	(*-------------- Services Stand EtherCAT Slave Faults----------------------------*)
	(*Fault584 - EtherCAT Slave Fault on Services Stand 01*)
		Fault_Tmrs[584].PT:= No_Timer;
		Fault_Tmrs[584]();
		Fault_Tmrs[584].IN:= GTAC_CONFIG.Option_Air1 AND NOT MAIN.SS01.DiscreteNode_OK;
		Out_To_ICxx.System_Faults[584]:=Fault_Tmrs[584].Q;
	(*Fault585 - EtherCAT Slave Fault on Services Stand 02*)
		Fault_Tmrs[585].PT:= No_Timer;
		Fault_Tmrs[585]();
		Fault_Tmrs[585].IN:= GTAC_CONFIG.Option_Air2 AND NOT MAIN.SS02.DiscreteNode_OK;
		Out_To_ICxx.System_Faults[585]:=Fault_Tmrs[585].Q;
	(*Fault586 - EtherCAT Slave Fault on Services Stand 03*)
		Fault_Tmrs[586].PT:= No_Timer;
		Fault_Tmrs[586]();
		Fault_Tmrs[586].IN:= FALSE AND NOT MAIN.SS03.DiscreteNode_OK;
		Out_To_ICxx.System_Faults[586]:=Fault_Tmrs[586].Q;

	(*-------------- Enable Switch Plate EtherCAT Slave Faults----------------------------*)
	(*Fault587 - EtherCAT Slave Fault on Enable Switch Plate 01*)
		Fault_Tmrs[587].PT:= No_Timer;
		Fault_Tmrs[587]();
		Fault_Tmrs[587].IN:= (GTAC_CONFIG.Option_ESW_Count>=1)
							AND NOT MAIN.ESW01.DiscreteNode_OK;
		Out_To_ICxx.System_Faults[587]:=Fault_Tmrs[587].Q;

	(*Fault588 - EtherCAT Slave Fault on Enable Switch Plate 02*)
		Fault_Tmrs[588].PT:= No_Timer;
		Fault_Tmrs[588]();
		Fault_Tmrs[588].IN:=  (GTAC_CONFIG.Option_ESW_Count>=2)
							 AND NOT MAIN.ESW02.DiscreteNode_OK;
		Out_To_ICxx.System_Faults[588]:=Fault_Tmrs[588].Q;

	(*Fault589 - EtherCAT Slave Fault on Enable Switch Plate 03*)
		Fault_Tmrs[589].PT:= No_Timer;
		Fault_Tmrs[589]();
		Fault_Tmrs[589].IN:=  (GTAC_CONFIG.Option_ESW_Count>=3)
							 AND NOT MAIN.ESW03.DiscreteNode_OK;
		Out_To_ICxx.System_Faults[589]:=Fault_Tmrs[589].Q;

	(*Fault590 - EtherCAT Slave Fault on Enable Switch Plate 04*)
		Fault_Tmrs[590].PT:= No_Timer;
		Fault_Tmrs[590]();
		Fault_Tmrs[590].IN:=  (GTAC_CONFIG.Option_ESW_Count>=4)
							 AND NOT MAIN.ESW04.DiscreteNode_OK;
		Out_To_ICxx.System_Faults[590]:=Fault_Tmrs[590].Q;

	(*-----------------ICxx EtherCAT Slave Faulted--------------*)

	(*Fault591 - EtherCAT Slave Fault In IC01 Cabinet*)
		Fault_Tmrs[591].PT:= No_Timer;
		Fault_Tmrs[591]();
		Fault_Tmrs[591].IN:= (GTAC_CONFIG.Option_IC_Count>=1) AND
							NOT MAIN.IC01.DiscreteNode_OK;
		Out_To_ICxx.System_Faults[591]:=Fault_Tmrs[591].Q;
	(*Fault592 - EtherCAT Slave Fault In IC02 Cabinet*)
		Fault_Tmrs[592].PT:= No_Timer;
		Fault_Tmrs[592]();
		Fault_Tmrs[592].IN:= (GTAC_CONFIG.Option_IC_Count>=2) AND
							NOT MAIN.IC02.DiscreteNode_OK;
		Out_To_ICxx.System_Faults[592]:=Fault_Tmrs[592].Q;
	(*Fault593 - EtherCAT Slave Fault In IC03 Cabinet*)
		Fault_Tmrs[593].PT:= No_Timer;
		Fault_Tmrs[593]();
		Fault_Tmrs[593].IN:= (GTAC_CONFIG.Option_IC_Count>=3) AND
							NOT MAIN.IC03.DiscreteNode_OK;
		Out_To_ICxx.System_Faults[593]:=Fault_Tmrs[593].Q;
	(*Fault594 - EtherCAT Slave Fault In IC04 Cabinet*)
		Fault_Tmrs[594].PT:= No_Timer;
		Fault_Tmrs[594]();
		Fault_Tmrs[594].IN:= (GTAC_CONFIG.Option_IC_Count>=4) AND
							NOT MAIN.IC04.DiscreteNode_OK;
		Out_To_ICxx.System_Faults[594]:=Fault_Tmrs[594].Q;
	(*Fault595 - EtherCAT Slave Fault In IC05 Cabinet*)
		Fault_Tmrs[595].PT:= No_Timer;
		Fault_Tmrs[595]();
		Fault_Tmrs[595].IN:= (GTAC_CONFIG.Option_IC_Count>=5) AND
							NOT MAIN.IC05.DiscreteNode_OK;
		Out_To_ICxx.System_Faults[595]:=Fault_Tmrs[595].Q;
	(*Fault596 - EtherCAT Slave Fault In IC06 Cabinet*)
		Fault_Tmrs[596].PT:= No_Timer;
		Fault_Tmrs[596]();
		Fault_Tmrs[596].IN:= (GTAC_CONFIG.Option_IC_Count>=6) AND
							NOT MAIN.IC06.DiscreteNode_OK;
		Out_To_ICxx.System_Faults[596]:=Fault_Tmrs[596].Q;
	(*Fault597 - EtherCAT Slave Fault In IC07 Cabinet*)
		Fault_Tmrs[597].PT:= No_Timer;
		Fault_Tmrs[597]();
		Fault_Tmrs[597].IN:= (GTAC_CONFIG.Option_IC_Count>=7) AND
							NOT MAIN.IC07.DiscreteNode_OK;
		Out_To_ICxx.System_Faults[597]:=Fault_Tmrs[597].Q;
	(*Fault598 - EtherCAT Slave Fault In IC08 Cabinet*)
		Fault_Tmrs[598].PT:= No_Timer;
		Fault_Tmrs[598]();
		Fault_Tmrs[598].IN:= (GTAC_CONFIG.Option_IC_Count>=8) AND
							NOT MAIN.IC08.DiscreteNode_OK;
		Out_To_ICxx.System_Faults[598]:=Fault_Tmrs[598].Q;

	(*------------------------------------------------- Fix_XX EtherCAT Slave Faults --------------------------------------------------*)

	(*IC related Fixtures (Human)*)
	(*Fault601 - EtherCAT Slave Fault On Fix at IC01.OP1*)
		Fault_Tmrs[601].PT:= No_Timer;
		Fault_Tmrs[601]();
		Fault_Tmrs[601].IN:= GTAC_CONFIG.Option_HumanFix_Enables.1 AND
							NOT Fix01.DiscreteNode_OK;
		Out_To_ICxx.System_Faults[601]:=Fault_Tmrs[601].Q;
	(*Fault602 - EtherCAT Slave Fault On Fix at IC01.OP2*)
		Fault_Tmrs[602].PT:= No_Timer;
		Fault_Tmrs[602]();
		Fault_Tmrs[602].IN:= GTAC_CONFIG.Option_HumanFix_Enables.2 AND
							NOT Fix02.DiscreteNode_OK;
		Out_To_ICxx.System_Faults[602]:=Fault_Tmrs[602].Q;

	(*Fault603 - EtherCAT Slave Fault On Fix at IC02.OP1*)
		Fault_Tmrs[603].PT:= No_Timer;
		Fault_Tmrs[603]();
		Fault_Tmrs[603].IN:= GTAC_CONFIG.Option_HumanFix_Enables.3 AND
							NOT Fix03.DiscreteNode_OK;
		Out_To_ICxx.System_Faults[603]:=Fault_Tmrs[603].Q;
	(*Fault604 - EtherCAT Slave Fault On Fix at IC02.OP2*)
		Fault_Tmrs[604].PT:= No_Timer;
		Fault_Tmrs[604]();
		Fault_Tmrs[604].IN:= GTAC_CONFIG.Option_HumanFix_Enables.4 AND
							NOT Fix04.DiscreteNode_OK;
		Out_To_ICxx.System_Faults[604]:=Fault_Tmrs[604].Q;

	(*Fault605 - EtherCAT Slave Fault On Fix at IC03.OP1*)
		Fault_Tmrs[605].PT:= No_Timer;
		Fault_Tmrs[605]();
		Fault_Tmrs[605].IN:= GTAC_CONFIG.Option_HumanFix_Enables.5 AND
							NOT Fix05.DiscreteNode_OK;
		Out_To_ICxx.System_Faults[605]:=Fault_Tmrs[605].Q;
	(*Fault606 - EtherCAT Slave Fault On Fix at IC03.OP2*)
		Fault_Tmrs[606].PT:= No_Timer;
		Fault_Tmrs[606]();
		Fault_Tmrs[606].IN:= GTAC_CONFIG.Option_HumanFix_Enables.6 AND
							NOT Fix06.DiscreteNode_OK;
		Out_To_ICxx.System_Faults[606]:=Fault_Tmrs[606].Q;

	(*Fault607 - EtherCAT Slave Fault On Fix at IC04.OP1*)
		Fault_Tmrs[607].PT:= No_Timer;
		Fault_Tmrs[607]();
		Fault_Tmrs[607].IN:= GTAC_CONFIG.Option_HumanFix_Enables.7 AND
							NOT Fix07.DiscreteNode_OK;
		Out_To_ICxx.System_Faults[607]:=Fault_Tmrs[607].Q;
	(*Fault608 - EtherCAT Slave Fault On Fix at IC04.OP2*)
		Fault_Tmrs[608].PT:= No_Timer;
		Fault_Tmrs[608]();
		Fault_Tmrs[608].IN:= GTAC_CONFIG.Option_HumanFix_Enables.8 AND
							NOT Fix08.DiscreteNode_OK;
		Out_To_ICxx.System_Faults[608]:=Fault_Tmrs[608].Q;

	(*Fault609 - EtherCAT Slave Fault On Fix at IC05.OP1*)
		Fault_Tmrs[609].PT:= No_Timer;
		Fault_Tmrs[609]();
		Fault_Tmrs[609].IN:= GTAC_CONFIG.Option_HumanFix_Enables.9 AND
							NOT Fix09.DiscreteNode_OK;
		Out_To_ICxx.System_Faults[609]:=Fault_Tmrs[609].Q;
	(*Fault610 - EtherCAT Slave Fault On Fix at IC05.OP2*)
		Fault_Tmrs[610].PT:= No_Timer;
		Fault_Tmrs[610]();
		Fault_Tmrs[610].IN:= GTAC_CONFIG.Option_HumanFix_Enables.10 AND
							NOT Fix10.DiscreteNode_OK;
		Out_To_ICxx.System_Faults[610]:=Fault_Tmrs[610].Q;

	(*Fault611 - EtherCAT Slave Fault On Fix at IC06.OP1*)
		Fault_Tmrs[611].PT:= No_Timer;
		Fault_Tmrs[611]();
		Fault_Tmrs[611].IN:= GTAC_CONFIG.Option_HumanFix_Enables.11 AND
							 NOT Fix11.DiscreteNode_OK;
		Out_To_ICxx.System_Faults[611]:=Fault_Tmrs[611].Q;
	(*Fault612 - EtherCAT Slave Fault On Fix at IC06.OP2*)
		Fault_Tmrs[612].PT:= No_Timer;
		Fault_Tmrs[612]();
		Fault_Tmrs[612].IN:= GTAC_CONFIG.Option_HumanFix_Enables.12 AND
							NOT Fix12.DiscreteNode_OK;
		Out_To_ICxx.System_Faults[612]:=Fault_Tmrs[612].Q;

	(*Fault613 - EtherCAT Slave Fault On Fix at IC07.OP1*)
		Fault_Tmrs[613].PT:= No_Timer;
		Fault_Tmrs[613]();
		Fault_Tmrs[613].IN:= GTAC_CONFIG.Option_HumanFix_Enables.13 AND
							NOT Fix13.DiscreteNode_OK;
		Out_To_ICxx.System_Faults[613]:=Fault_Tmrs[613].Q;
	(*Fault614 - EtherCAT Slave Fault On Fix at IC07.OP2*)
		Fault_Tmrs[614].PT:= No_Timer;
		Fault_Tmrs[614]();
		Fault_Tmrs[614].IN:= GTAC_CONFIG.Option_HumanFix_Enables.14 AND
							NOT Fix14.DiscreteNode_OK;
		Out_To_ICxx.System_Faults[614]:=Fault_Tmrs[614].Q;

	(*Fault615 - EtherCAT Slave Fault On Fix at IC08.OP1*)
		Fault_Tmrs[615].PT:= No_Timer;
		Fault_Tmrs[615]();
		Fault_Tmrs[615].IN:= GTAC_CONFIG.Option_HumanFix_Enables.15 AND
							NOT Fix15.DiscreteNode_OK;
		Out_To_ICxx.System_Faults[615]:=Fault_Tmrs[615].Q;
	(*Fault616 - EtherCAT Slave Fault On Fix at IC08.OP2*)
		Fault_Tmrs[616].PT:= No_Timer;
		Fault_Tmrs[616]();
		Fault_Tmrs[616].IN:= GTAC_CONFIG.Option_HumanFix_Enables.16 AND
							NOT Fix16.DiscreteNode_OK;
		Out_To_ICxx.System_Faults[616]:=Fault_Tmrs[616].Q;

	(*Internal Fixtures*)
	(*Fault617 - EtherCAT Slave Fault On Internal Fix 101*)
		Fault_Tmrs[617].PT:= No_Timer;
		Fault_Tmrs[617]();
		Fault_Tmrs[617].IN:= (GTAC_CONFIG.Option_InternalFix_Count>=1) AND
							NOT Fix101.DiscreteNode_OK;
		Out_To_ICxx.System_Faults[617]:=Fault_Tmrs[617].Q;

	(*Fault618 - EtherCAT Slave Fault On Internal Fix 102*)
		Fault_Tmrs[618].PT:= No_Timer;
		Fault_Tmrs[618]();
		Fault_Tmrs[618].IN:= (GTAC_CONFIG.Option_InternalFix_Count>=2) AND
							NOT Fix102.DiscreteNode_OK;
		Out_To_ICxx.System_Faults[618]:=Fault_Tmrs[618].Q;

	(*Fault619 - EtherCAT Slave Fault On Internal Fix 103*)
		Fault_Tmrs[619].PT:= No_Timer;
		Fault_Tmrs[619]();
		Fault_Tmrs[619].IN:= (GTAC_CONFIG.Option_InternalFix_Count>=3) AND
							NOT Fix103.DiscreteNode_OK;
		Out_To_ICxx.System_Faults[619]:=Fault_Tmrs[619].Q;

	(*Fault620 - EtherCAT Slave Fault On Internal Fix 104*)
		Fault_Tmrs[620].PT:= No_Timer;
		Fault_Tmrs[620]();
		Fault_Tmrs[620].IN:= (GTAC_CONFIG.Option_InternalFix_Count>=4) AND
							NOT Fix104.DiscreteNode_OK;
		Out_To_ICxx.System_Faults[620]:=Fault_Tmrs[620].Q;

	(*Fault621 - EtherCAT Slave Fault On Internal Fix 105*)
		Fault_Tmrs[621].PT:= No_Timer;
		Fault_Tmrs[621]();
		Fault_Tmrs[621].IN:= (GTAC_CONFIG.Option_InternalFix_Count>=5) AND
							NOT Fix105.DiscreteNode_OK;
		Out_To_ICxx.System_Faults[621]:=Fault_Tmrs[621].Q;

	(*Fault622 - EtherCAT Slave Fault On Internal Fix 106*)
		Fault_Tmrs[622].PT:= No_Timer;
		Fault_Tmrs[622]();
		Fault_Tmrs[622].IN:= (GTAC_CONFIG.Option_InternalFix_Count>=6) AND
							NOT Fix106.DiscreteNode_OK;
		Out_To_ICxx.System_Faults[622]:=Fault_Tmrs[622].Q;

	(*Fault623 - EtherCAT Slave Fault On Internal Fix 107*)
		Fault_Tmrs[623].PT:= No_Timer;
		Fault_Tmrs[623]();
		Fault_Tmrs[623].IN:= (GTAC_CONFIG.Option_InternalFix_Count>=7) AND
							NOT Fix107.DiscreteNode_OK;
		Out_To_ICxx.System_Faults[623]:=Fault_Tmrs[623].Q;

	(*Fault624 - EtherCAT Slave Fault On Internal Fix 108*)
		Fault_Tmrs[624].PT:= No_Timer;
		Fault_Tmrs[624]();
		Fault_Tmrs[624].IN:= (GTAC_CONFIG.Option_InternalFix_Count>=8) AND
							NOT Fix108.DiscreteNode_OK;
		Out_To_ICxx.System_Faults[624]:=Fault_Tmrs[624].Q;

	(*Fault625 - EtherCAT Slave Fault On Internal Fix 109*)
		Fault_Tmrs[625].PT:= No_Timer;
		Fault_Tmrs[625]();
		Fault_Tmrs[625].IN:= (GTAC_CONFIG.Option_InternalFix_Count>=9) AND
							NOT Fix109.DiscreteNode_OK;
		Out_To_ICxx.System_Faults[625]:=Fault_Tmrs[625].Q;

	(*Fault626 - EtherCAT Slave Fault On Internal Fix 110*)
		Fault_Tmrs[626].PT:= No_Timer;
		Fault_Tmrs[626]();
		Fault_Tmrs[626].IN:= (GTAC_CONFIG.Option_InternalFix_Count>=10) AND
							NOT Fix110.DiscreteNode_OK;
		Out_To_ICxx.System_Faults[626]:=Fault_Tmrs[626].Q;

	(*Fault627 - EtherCAT Slave Fault On Internal Fix 111*)
		Fault_Tmrs[627].PT:= No_Timer;
		Fault_Tmrs[627]();
		Fault_Tmrs[627].IN:= (GTAC_CONFIG.Option_InternalFix_Count>=11) AND
							NOT Fix111.DiscreteNode_OK;
		Out_To_ICxx.System_Faults[627]:=Fault_Tmrs[627].Q;

	(*Fault628 - EtherCAT Slave Fault On Internal Fix 112*)
		Fault_Tmrs[628].PT:= No_Timer;
		Fault_Tmrs[628]();
		Fault_Tmrs[628].IN:= (GTAC_CONFIG.Option_InternalFix_Count>=12) AND
							NOT Fix112.DiscreteNode_OK;
		Out_To_ICxx.System_Faults[628]:=Fault_Tmrs[628].Q;


	(*-----------------Rxx EtherCAT Slave Faulted--------------*)

	(*Fault631 - EtherCAT Slave Fault In R1 Cabinet*)
		Fault_Tmrs[631].PT:= No_Timer;
		Fault_Tmrs[631]();
		Fault_Tmrs[631].IN:= (GTAC_CONFIG.Option_Robot_Count>=1)  AND
							NOT MAIN.R1.DiscreteNode_OK;
		Out_To_ICxx.System_Faults[631]:=Fault_Tmrs[631].Q;
	(*Fault632 - EtherCAT Slave Fault In R2 Cabinet*)
		Fault_Tmrs[632].PT:= No_Timer;
		Fault_Tmrs[632]();
		Fault_Tmrs[632].IN:= (GTAC_CONFIG.Option_Robot_Count>=2)  AND
							NOT MAIN.R2.DiscreteNode_OK;
		Out_To_ICxx.System_Faults[632]:=Fault_Tmrs[632].Q;
	(*Fault633 - EtherCAT Slave Fault In R3 Cabinet*)
		Fault_Tmrs[633].PT:= No_Timer;
		Fault_Tmrs[633]();
		Fault_Tmrs[633].IN:= (GTAC_CONFIG.Option_Robot_Count>=3)  AND
							NOT MAIN.R3.DiscreteNode_OK;
		Out_To_ICxx.System_Faults[633]:=Fault_Tmrs[633].Q;
	(*Fault634 - EtherCAT Slave Fault In R4 Cabinet*)
		Fault_Tmrs[634].PT:= No_Timer;
		Fault_Tmrs[634]();
		Fault_Tmrs[634].IN:= (GTAC_CONFIG.Option_Robot_Count>=4)  AND
							NOT MAIN.R4.DiscreteNode_OK;
		Out_To_ICxx.System_Faults[634]:=Fault_Tmrs[634].Q;
	(*Fault635 - EtherCAT Slave Fault In R5 Cabinet*)
		Fault_Tmrs[635].PT:= No_Timer;
		Fault_Tmrs[635]();
		Fault_Tmrs[635].IN:= (GTAC_CONFIG.Option_Robot_Count>=5)  AND
							NOT MAIN.R5.DiscreteNode_OK;
		Out_To_ICxx.System_Faults[635]:=Fault_Tmrs[635].Q;
	(*Fault636 - EtherCAT Slave Fault In R6 Cabinet*)
		Fault_Tmrs[636].PT:= No_Timer;
		Fault_Tmrs[636]();
		Fault_Tmrs[636].IN:= (GTAC_CONFIG.Option_Robot_Count>=6)  AND
							NOT MAIN.R6.DiscreteNode_OK;
		Out_To_ICxx.System_Faults[636]:=Fault_Tmrs[636].Q;
	(*Fault637 - EtherCAT Slave Fault In R7 Cabinet*)
		Fault_Tmrs[637].PT:= No_Timer;
		Fault_Tmrs[637]();
		Fault_Tmrs[637].IN:= (GTAC_CONFIG.Option_Robot_Count>=7)  AND
							NOT MAIN.R7.DiscreteNode_OK;
		Out_To_ICxx.System_Faults[637]:=Fault_Tmrs[637].Q;
	(*Fault638 - EtherCAT Slave Fault In R8 Cabinet*)
		Fault_Tmrs[638].PT:= No_Timer;
		Fault_Tmrs[638]();
		Fault_Tmrs[638].IN:= (GTAC_CONFIG.Option_Robot_Count>=8)  AND
							NOT MAIN.R8.DiscreteNode_OK;
		Out_To_ICxx.System_Faults[638]:=Fault_Tmrs[638].Q;
	(*Fault639 - EtherCAT Slave Fault In R9 Cabinet*)
		Fault_Tmrs[639].PT:= No_Timer;
		Fault_Tmrs[639]();
		Fault_Tmrs[639].IN:= (GTAC_CONFIG.Option_Robot_Count>=9)  AND
							NOT MAIN.R9.DiscreteNode_OK;
		Out_To_ICxx.System_Faults[639]:=Fault_Tmrs[639].Q;
	(*Fault640 - EtherCAT Slave Fault In R10 Cabinet*)
		Fault_Tmrs[640].PT:= No_Timer;
		Fault_Tmrs[640]();
		Fault_Tmrs[640].IN:= (GTAC_CONFIG.Option_Robot_Count>=10)  AND
							NOT MAIN.R10.DiscreteNode_OK;
		Out_To_ICxx.System_Faults[640]:=Fault_Tmrs[640].Q;
	(*Fault641 - EtherCAT Slave Fault In R11 Cabinet*)
		Fault_Tmrs[641].PT:= No_Timer;
		Fault_Tmrs[641]();
		Fault_Tmrs[641].IN:= (GTAC_CONFIG.Option_Robot_Count>=11)  AND
							NOT MAIN.R11.DiscreteNode_OK;
		Out_To_ICxx.System_Faults[641]:=Fault_Tmrs[641].Q;
	(*Fault642 - EtherCAT Slave Fault In R12 Cabinet*)
		Fault_Tmrs[642].PT:= No_Timer;
		Fault_Tmrs[642]();
		Fault_Tmrs[642].IN:= (GTAC_CONFIG.Option_Robot_Count>=12)  AND
							NOT MAIN.R12.DiscreteNode_OK;
		Out_To_ICxx.System_Faults[642]:=Fault_Tmrs[642].Q;
	(*Fault643 - EtherCAT Slave Fault In R13 Cabinet*)
		Fault_Tmrs[643].PT:= No_Timer;
		Fault_Tmrs[643]();
		Fault_Tmrs[643].IN:= (GTAC_CONFIG.Option_Robot_Count>=13)  AND
							NOT MAIN.R13.DiscreteNode_OK;
		Out_To_ICxx.System_Faults[643]:=Fault_Tmrs[643].Q;
	(*Fault644 - EtherCAT Slave Fault In R14 Cabinet*)
		Fault_Tmrs[644].PT:= No_Timer;
		Fault_Tmrs[644]();
		Fault_Tmrs[644].IN:= (GTAC_CONFIG.Option_Robot_Count>=14)  AND
							NOT MAIN.R14.DiscreteNode_OK;
		Out_To_ICxx.System_Faults[644]:=Fault_Tmrs[644].Q;
	(*Fault645 - EtherCAT Slave Fault In R15 Cabinet*)
		Fault_Tmrs[645].PT:= No_Timer;
		Fault_Tmrs[645]();
		Fault_Tmrs[645].IN:= (GTAC_CONFIG.Option_Robot_Count>=15)  AND
							NOT MAIN.R15.DiscreteNode_OK;
		Out_To_ICxx.System_Faults[645]:=Fault_Tmrs[645].Q;
	(*Fault646 - EtherCAT Slave Fault In R16 Cabinet*)
		Fault_Tmrs[646].PT:= No_Timer;
		Fault_Tmrs[646]();
		Fault_Tmrs[646].IN:= (GTAC_CONFIG.Option_Robot_Count>=16)  AND
							NOT MAIN.R16.DiscreteNode_OK;
		Out_To_ICxx.System_Faults[646]:=Fault_Tmrs[646].Q;
	(*Fault647 - EtherCAT Slave Fault In R17 Cabinet*)
		Fault_Tmrs[647].PT:= No_Timer;
		Fault_Tmrs[647]();
		Fault_Tmrs[647].IN:= (GTAC_CONFIG.Option_Robot_Count>=17)  AND
							NOT MAIN.R17.DiscreteNode_OK;
		Out_To_ICxx.System_Faults[647]:=Fault_Tmrs[647].Q;
	(*Fault648 - EtherCAT Slave Fault In R18 Cabinet*)
		Fault_Tmrs[648].PT:= No_Timer;
		Fault_Tmrs[648]();
		Fault_Tmrs[648].IN:= (GTAC_CONFIG.Option_Robot_Count>=18)  AND
							NOT MAIN.R18.DiscreteNode_OK;
		Out_To_ICxx.System_Faults[648]:=Fault_Tmrs[648].Q;
	(*Fault649 - EtherCAT Slave Fault In R19 Cabinet*)
		Fault_Tmrs[649].PT:= No_Timer;
		Fault_Tmrs[649]();
		Fault_Tmrs[649].IN:= (GTAC_CONFIG.Option_Robot_Count>=19)  AND
							NOT MAIN.R19.DiscreteNode_OK;
		Out_To_ICxx.System_Faults[649]:=Fault_Tmrs[649].Q;
	(*Fault650 - EtherCAT Slave Fault In R20 Cabinet*)
		Fault_Tmrs[650].PT:= No_Timer;
		Fault_Tmrs[650]();
		Fault_Tmrs[650].IN:= (GTAC_CONFIG.Option_Robot_Count>=20)  AND
							NOT MAIN.R20.DiscreteNode_OK;
		Out_To_ICxx.System_Faults[650]:=Fault_Tmrs[650].Q;
	(*Fault651 - EtherCAT Slave Fault In R21 Cabinet*)
		Fault_Tmrs[651].PT:= No_Timer;
		Fault_Tmrs[651]();
		Fault_Tmrs[651].IN:= (GTAC_CONFIG.Option_Robot_Count>=21)  AND
							NOT MAIN.R21.DiscreteNode_OK;
		Out_To_ICxx.System_Faults[651]:=Fault_Tmrs[651].Q;
	(*Fault652 - EtherCAT Slave Fault In R22 Cabinet*)
		Fault_Tmrs[652].PT:= No_Timer;
		Fault_Tmrs[652]();
		Fault_Tmrs[652].IN:= (GTAC_CONFIG.Option_Robot_Count>=22)  AND
							NOT MAIN.R22.DiscreteNode_OK;
		Out_To_ICxx.System_Faults[652]:=Fault_Tmrs[652].Q;
	(*Fault653 - EtherCAT Slave Fault In R23 Cabinet*)
		Fault_Tmrs[653].PT:= No_Timer;
		Fault_Tmrs[653]();
		Fault_Tmrs[653].IN:= (GTAC_CONFIG.Option_Robot_Count>=23)  AND
							NOT MAIN.R23.DiscreteNode_OK;
		Out_To_ICxx.System_Faults[653]:=Fault_Tmrs[653].Q;
	(*Fault654 - EtherCAT Slave Fault In R24 Cabinet*)
		Fault_Tmrs[654].PT:= No_Timer;
		Fault_Tmrs[654]();
		Fault_Tmrs[654].IN:= (GTAC_CONFIG.Option_Robot_Count>=24)  AND
							NOT MAIN.R24.DiscreteNode_OK;
		Out_To_ICxx.System_Faults[654]:=Fault_Tmrs[654].Q;
	(*Fault655 - EtherCAT Slave Fault In R25 Cabinet*)
		Fault_Tmrs[655].PT:= No_Timer;
		Fault_Tmrs[655]();
		Fault_Tmrs[655].IN:= (GTAC_CONFIG.Option_Robot_Count>=25)  AND
							NOT MAIN.R25.DiscreteNode_OK;
		Out_To_ICxx.System_Faults[655]:=Fault_Tmrs[655].Q;
	(*Fault656 - EtherCAT Slave Fault In R26 Cabinet*)
		Fault_Tmrs[656].PT:= No_Timer;
		Fault_Tmrs[656]();
		Fault_Tmrs[656].IN:= (GTAC_CONFIG.Option_Robot_Count>=26)  AND
							NOT MAIN.R26.DiscreteNode_OK;
		Out_To_ICxx.System_Faults[656]:=Fault_Tmrs[656].Q;
	(*Fault657 - EtherCAT Slave Fault In R27 Cabinet*)
		Fault_Tmrs[657].PT:= No_Timer;
		Fault_Tmrs[657]();
		Fault_Tmrs[657].IN:= (GTAC_CONFIG.Option_Robot_Count>=27)  AND
							NOT MAIN.R27.DiscreteNode_OK;
		Out_To_ICxx.System_Faults[657]:=Fault_Tmrs[657].Q;
	(*Fault658 - EtherCAT Slave Fault In R28 Cabinet*)
		Fault_Tmrs[658].PT:= No_Timer;
		Fault_Tmrs[658]();
		Fault_Tmrs[658].IN:= (GTAC_CONFIG.Option_Robot_Count>=28)  AND
							NOT MAIN.R28.DiscreteNode_OK;
		Out_To_ICxx.System_Faults[658]:=Fault_Tmrs[658].Q;
	(*Fault659 - EtherCAT Slave Fault In R29 Cabinet*)
		Fault_Tmrs[659].PT:= No_Timer;
		Fault_Tmrs[659]();
		Fault_Tmrs[659].IN:= (GTAC_CONFIG.Option_Robot_Count>=29)  AND
							NOT MAIN.R29.DiscreteNode_OK;
		Out_To_ICxx.System_Faults[659]:=Fault_Tmrs[659].Q;
	(*Fault660 - EtherCAT Slave Fault In R30 Cabinet*)
		Fault_Tmrs[660].PT:= No_Timer;
		Fault_Tmrs[660]();
		Fault_Tmrs[660].IN:= (GTAC_CONFIG.Option_Robot_Count>=30)  AND
							NOT MAIN.R30.DiscreteNode_OK;
		Out_To_ICxx.System_Faults[660]:=Fault_Tmrs[660].Q;

	(*-----------------Rxx Water Stand EtherCAT Slave Faulted--------------*)

	(*Fault661 - EtherCAT Slave Fault On R1 Water Stand*)
		Fault_Tmrs[661].PT:= No_Timer;
		Fault_Tmrs[661]();
		Fault_Tmrs[661].IN:= (GTAC_CONFIG.Option_Robot_Count>=1)  AND
							(((MAIN.R1.FB_In.Options.WaterStand_Amount>0) AND
							NOT MAIN.R1.WS[1].DiscreteNode_OK) OR
							((MAIN.R1.FB_In.Options.WaterStand_Amount>1) AND
							NOT MAIN.R1.WS[2].DiscreteNode_OK));
		Out_To_ICxx.System_Faults[661]:=Fault_Tmrs[661].Q;
	(*Fault662 - EtherCAT Slave Fault On R2 Water Stand*)
		Fault_Tmrs[662].PT:= No_Timer;
		Fault_Tmrs[662]();
		Fault_Tmrs[662].IN:= (GTAC_CONFIG.Option_Robot_Count>=2)  AND
							(((MAIN.R2.FB_In.Options.WaterStand_Amount>0) AND
							NOT MAIN.R2.WS[1].DiscreteNode_OK) OR
							((MAIN.R2.FB_In.Options.WaterStand_Amount>1) AND
							NOT MAIN.R2.WS[2].DiscreteNode_OK));
		Out_To_ICxx.System_Faults[662]:=Fault_Tmrs[662].Q;
	(*Fault663 - EtherCAT Slave Fault On R3 Water Stand*)
		Fault_Tmrs[663].PT:= No_Timer;
		Fault_Tmrs[663]();
		Fault_Tmrs[663].IN:= (GTAC_CONFIG.Option_Robot_Count>=3)  AND
							(((MAIN.R3.FB_In.Options.WaterStand_Amount>0) AND
							NOT MAIN.R3.WS[1].DiscreteNode_OK) OR
							((MAIN.R3.FB_In.Options.WaterStand_Amount>1) AND
							NOT MAIN.R3.WS[2].DiscreteNode_OK));
		Out_To_ICxx.System_Faults[663]:=Fault_Tmrs[663].Q;
	(*Fault664 - EtherCAT Slave Fault On R4 Water Stand*)
		Fault_Tmrs[664].PT:= No_Timer;
		Fault_Tmrs[664]();
		Fault_Tmrs[664].IN:= (GTAC_CONFIG.Option_Robot_Count>=4)  AND
							(((MAIN.R4.FB_In.Options.WaterStand_Amount>0) AND
							NOT MAIN.R4.WS[1].DiscreteNode_OK) OR
							((MAIN.R4.FB_In.Options.WaterStand_Amount>1) AND
							NOT MAIN.R4.WS[2].DiscreteNode_OK));
		Out_To_ICxx.System_Faults[664]:=Fault_Tmrs[664].Q;
	(*Fault665 - EtherCAT Slave Fault On R5 Water Stand*)
		Fault_Tmrs[665].PT:= No_Timer;
		Fault_Tmrs[665]();
		Fault_Tmrs[665].IN:= (GTAC_CONFIG.Option_Robot_Count>=5)  AND
							(((MAIN.R5.FB_In.Options.WaterStand_Amount>0) AND
							NOT MAIN.R5.WS[1].DiscreteNode_OK) OR
							((MAIN.R5.FB_In.Options.WaterStand_Amount>1) AND
							NOT MAIN.R5.WS[2].DiscreteNode_OK));
		Out_To_ICxx.System_Faults[665]:=Fault_Tmrs[665].Q;
	(*Fault666 - EtherCAT Slave Fault On R6 Water Stand*)
		Fault_Tmrs[666].PT:= No_Timer;
		Fault_Tmrs[666]();
		Fault_Tmrs[666].IN:= (GTAC_CONFIG.Option_Robot_Count>=6)  AND
							(((MAIN.R6.FB_In.Options.WaterStand_Amount>0) AND
							NOT MAIN.R6.WS[1].DiscreteNode_OK) OR
							((MAIN.R6.FB_In.Options.WaterStand_Amount>1) AND
							NOT MAIN.R6.WS[2].DiscreteNode_OK));
		Out_To_ICxx.System_Faults[666]:=Fault_Tmrs[666].Q;
	(*Fault667 - EtherCAT Slave Fault On R7 Water Stand*)
		Fault_Tmrs[667].PT:= No_Timer;
		Fault_Tmrs[667]();
		Fault_Tmrs[667].IN:= (GTAC_CONFIG.Option_Robot_Count>=7)  AND
							(((MAIN.R7.FB_In.Options.WaterStand_Amount>0) AND
							NOT MAIN.R7.WS[1].DiscreteNode_OK) OR
							((MAIN.R7.FB_In.Options.WaterStand_Amount>1) AND
							NOT MAIN.R7.WS[2].DiscreteNode_OK));
		Out_To_ICxx.System_Faults[667]:=Fault_Tmrs[667].Q;
	(*Fault668 - EtherCAT Slave Fault On R8 Water Stand*)
		Fault_Tmrs[668].PT:= No_Timer;
		Fault_Tmrs[668]();
		Fault_Tmrs[668].IN:= (GTAC_CONFIG.Option_Robot_Count>=8)  AND
							(((MAIN.R8.FB_In.Options.WaterStand_Amount>0) AND
							NOT MAIN.R8.WS[1].DiscreteNode_OK) OR
							((MAIN.R8.FB_In.Options.WaterStand_Amount>1) AND
							NOT MAIN.R8.WS[2].DiscreteNode_OK));
		Out_To_ICxx.System_Faults[668]:=Fault_Tmrs[668].Q;
	(*Fault669 - EtherCAT Slave Fault On R9 Water Stand*)
		Fault_Tmrs[669].PT:= No_Timer;
		Fault_Tmrs[669]();
		Fault_Tmrs[669].IN:= (GTAC_CONFIG.Option_Robot_Count>=9)  AND
							(((MAIN.R9.FB_In.Options.WaterStand_Amount>0) AND
							NOT MAIN.R9.WS[1].DiscreteNode_OK) OR
							((MAIN.R9.FB_In.Options.WaterStand_Amount>1) AND
							NOT MAIN.R9.WS[2].DiscreteNode_OK));
		Out_To_ICxx.System_Faults[669]:=Fault_Tmrs[669].Q;
	(*Fault670 - EtherCAT Slave Fault On R10 Water Stand*)
		Fault_Tmrs[670].PT:= No_Timer;
		Fault_Tmrs[670]();
		Fault_Tmrs[670].IN:= (GTAC_CONFIG.Option_Robot_Count>=10)  AND
							(((MAIN.R10.FB_In.Options.WaterStand_Amount>0) AND
							NOT MAIN.R10.WS[1].DiscreteNode_OK) OR
							((MAIN.R10.FB_In.Options.WaterStand_Amount>1) AND
							NOT MAIN.R10.WS[2].DiscreteNode_OK));
		Out_To_ICxx.System_Faults[670]:=Fault_Tmrs[670].Q;
	(*Fault671 - EtherCAT Slave Fault On R11 Water Stand*)
		Fault_Tmrs[671].PT:= No_Timer;
		Fault_Tmrs[671]();
		Fault_Tmrs[671].IN:= (GTAC_CONFIG.Option_Robot_Count>=11)  AND
							(((MAIN.R11.FB_In.Options.WaterStand_Amount>0) AND
							NOT MAIN.R11.WS[1].DiscreteNode_OK) OR
							((MAIN.R11.FB_In.Options.WaterStand_Amount>1) AND
							NOT MAIN.R11.WS[2].DiscreteNode_OK));
		Out_To_ICxx.System_Faults[671]:=Fault_Tmrs[671].Q;
	(*Fault672 - EtherCAT Slave Fault On R12 Water Stand*)
		Fault_Tmrs[672].PT:= No_Timer;
		Fault_Tmrs[672]();
		Fault_Tmrs[672].IN:= (GTAC_CONFIG.Option_Robot_Count>=12)  AND
							(((MAIN.R12.FB_In.Options.WaterStand_Amount>0) AND
							NOT MAIN.R12.WS[1].DiscreteNode_OK) OR
							((MAIN.R12.FB_In.Options.WaterStand_Amount>1) AND
							NOT MAIN.R12.WS[2].DiscreteNode_OK));
		Out_To_ICxx.System_Faults[672]:=Fault_Tmrs[672].Q;
	(*Fault673 - EtherCAT Slave Fault On R13 Water Stand*)
		Fault_Tmrs[673].PT:= No_Timer;
		Fault_Tmrs[673]();
		Fault_Tmrs[673].IN:= (GTAC_CONFIG.Option_Robot_Count>=13)  AND
							(((MAIN.R13.FB_In.Options.WaterStand_Amount>0) AND
							NOT MAIN.R13.WS[1].DiscreteNode_OK) OR
							((MAIN.R13.FB_In.Options.WaterStand_Amount>1) AND
							NOT MAIN.R13.WS[2].DiscreteNode_OK));
		Out_To_ICxx.System_Faults[673]:=Fault_Tmrs[673].Q;
	(*Fault674 - EtherCAT Slave Fault On R14 Water Stand*)
		Fault_Tmrs[674].PT:= No_Timer;
		Fault_Tmrs[674]();
		Fault_Tmrs[674].IN:= (GTAC_CONFIG.Option_Robot_Count>=14)  AND
							(((MAIN.R14.FB_In.Options.WaterStand_Amount>0) AND
							NOT MAIN.R14.WS[1].DiscreteNode_OK) OR
							((MAIN.R14.FB_In.Options.WaterStand_Amount>1) AND
							NOT MAIN.R14.WS[2].DiscreteNode_OK));
		Out_To_ICxx.System_Faults[674]:=Fault_Tmrs[674].Q;
	(*Fault675 - EtherCAT Slave Fault On R15 Water Stand*)
		Fault_Tmrs[675].PT:= No_Timer;
		Fault_Tmrs[675]();
		Fault_Tmrs[675].IN:= (GTAC_CONFIG.Option_Robot_Count>=15)  AND
							(((MAIN.R15.FB_In.Options.WaterStand_Amount>0) AND
							NOT MAIN.R15.WS[1].DiscreteNode_OK) OR
							((MAIN.R15.FB_In.Options.WaterStand_Amount>1) AND
							NOT MAIN.R15.WS[2].DiscreteNode_OK));
		Out_To_ICxx.System_Faults[675]:=Fault_Tmrs[675].Q;
	(*Fault676 - EtherCAT Slave Fault On R16 Water Stand*)
		Fault_Tmrs[676].PT:= No_Timer;
		Fault_Tmrs[676]();
		Fault_Tmrs[676].IN:= (GTAC_CONFIG.Option_Robot_Count>=16)  AND
							(((MAIN.R16.FB_In.Options.WaterStand_Amount>0) AND
							NOT MAIN.R16.WS[1].DiscreteNode_OK) OR
							((MAIN.R16.FB_In.Options.WaterStand_Amount>1) AND
							NOT MAIN.R16.WS[2].DiscreteNode_OK));
		Out_To_ICxx.System_Faults[676]:=Fault_Tmrs[676].Q;
	(*Fault677 - EtherCAT Slave Fault On R17 Water Stand*)
		Fault_Tmrs[677].PT:= No_Timer;
		Fault_Tmrs[677]();
		Fault_Tmrs[677].IN:= (GTAC_CONFIG.Option_Robot_Count>=17)  AND
							(((MAIN.R17.FB_In.Options.WaterStand_Amount>0) AND
							NOT MAIN.R17.WS[1].DiscreteNode_OK) OR
							((MAIN.R17.FB_In.Options.WaterStand_Amount>1) AND
							NOT MAIN.R17.WS[2].DiscreteNode_OK));
		Out_To_ICxx.System_Faults[677]:=Fault_Tmrs[677].Q;
	(*Fault678 - EtherCAT Slave Fault On R18 Water Stand*)
		Fault_Tmrs[678].PT:= No_Timer;
		Fault_Tmrs[678]();
		Fault_Tmrs[678].IN:= (GTAC_CONFIG.Option_Robot_Count>=18)  AND
							(((MAIN.R18.FB_In.Options.WaterStand_Amount>0) AND
							NOT MAIN.R18.WS[1].DiscreteNode_OK) OR
							((MAIN.R18.FB_In.Options.WaterStand_Amount>1) AND
							NOT MAIN.R18.WS[2].DiscreteNode_OK));
		Out_To_ICxx.System_Faults[678]:=Fault_Tmrs[678].Q;
	(*Fault679 - EtherCAT Slave Fault On R19 Water Stand*)
		Fault_Tmrs[679].PT:= No_Timer;
		Fault_Tmrs[679]();
		Fault_Tmrs[679].IN:= (GTAC_CONFIG.Option_Robot_Count>=19)  AND
							(((MAIN.R19.FB_In.Options.WaterStand_Amount>0) AND
							NOT MAIN.R19.WS[1].DiscreteNode_OK) OR
							((MAIN.R19.FB_In.Options.WaterStand_Amount>1) AND
							NOT MAIN.R19.WS[2].DiscreteNode_OK));
		Out_To_ICxx.System_Faults[679]:=Fault_Tmrs[679].Q;
	(*Fault680 - EtherCAT Slave Fault On R20 Water Stand*)
		Fault_Tmrs[680].PT:= No_Timer;
		Fault_Tmrs[680]();
		Fault_Tmrs[680].IN:= (GTAC_CONFIG.Option_Robot_Count>=20)  AND
							(((MAIN.R20.FB_In.Options.WaterStand_Amount>0) AND
							NOT MAIN.R20.WS[1].DiscreteNode_OK) OR
							((MAIN.R20.FB_In.Options.WaterStand_Amount>1) AND
							NOT MAIN.R20.WS[2].DiscreteNode_OK));
		Out_To_ICxx.System_Faults[680]:=Fault_Tmrs[680].Q;
	(*Fault681 - EtherCAT Slave Fault On R21 Water Stand*)
		Fault_Tmrs[681].PT:= No_Timer;
		Fault_Tmrs[681]();
		Fault_Tmrs[681].IN:= (GTAC_CONFIG.Option_Robot_Count>=21)  AND
							(((MAIN.R21.FB_In.Options.WaterStand_Amount>0) AND
							NOT MAIN.R21.WS[1].DiscreteNode_OK) OR
							((MAIN.R21.FB_In.Options.WaterStand_Amount>1) AND
							NOT MAIN.R21.WS[2].DiscreteNode_OK));
		Out_To_ICxx.System_Faults[681]:=Fault_Tmrs[681].Q;
	(*Fault682 - EtherCAT Slave Fault On R22 Water Stand*)
		Fault_Tmrs[682].PT:= No_Timer;
		Fault_Tmrs[682]();
		Fault_Tmrs[682].IN:= (GTAC_CONFIG.Option_Robot_Count>=22)  AND
							(((MAIN.R22.FB_In.Options.WaterStand_Amount>0) AND
							NOT MAIN.R22.WS[1].DiscreteNode_OK) OR
							((MAIN.R22.FB_In.Options.WaterStand_Amount>1) AND
							NOT MAIN.R22.WS[2].DiscreteNode_OK));
		Out_To_ICxx.System_Faults[682]:=Fault_Tmrs[682].Q;
	(*Fault683 - EtherCAT Slave Fault On R23 Water Stand*)
		Fault_Tmrs[683].PT:= No_Timer;
		Fault_Tmrs[683]();
		Fault_Tmrs[683].IN:= (GTAC_CONFIG.Option_Robot_Count>=23)  AND
							(((MAIN.R23.FB_In.Options.WaterStand_Amount>0) AND
							NOT MAIN.R23.WS[1].DiscreteNode_OK) OR
							((MAIN.R23.FB_In.Options.WaterStand_Amount>1) AND
							NOT MAIN.R23.WS[2].DiscreteNode_OK));
		Out_To_ICxx.System_Faults[683]:=Fault_Tmrs[683].Q;
	(*Fault684 - EtherCAT Slave Fault On R24 Water Stand*)
		Fault_Tmrs[684].PT:= No_Timer;
		Fault_Tmrs[684]();
		Fault_Tmrs[684].IN:= (GTAC_CONFIG.Option_Robot_Count>=24)  AND
							(((MAIN.R24.FB_In.Options.WaterStand_Amount>0) AND
							NOT MAIN.R24.WS[1].DiscreteNode_OK) OR
							((MAIN.R24.FB_In.Options.WaterStand_Amount>1) AND
							NOT MAIN.R24.WS[2].DiscreteNode_OK));
		Out_To_ICxx.System_Faults[684]:=Fault_Tmrs[684].Q;
	(*Fault685 - EtherCAT Slave Fault On R25 Water Stand*)
		Fault_Tmrs[685].PT:= No_Timer;
		Fault_Tmrs[685]();
		Fault_Tmrs[685].IN:= (GTAC_CONFIG.Option_Robot_Count>=25)  AND
							(((MAIN.R25.FB_In.Options.WaterStand_Amount>0) AND
							NOT MAIN.R25.WS[1].DiscreteNode_OK) OR
							((MAIN.R25.FB_In.Options.WaterStand_Amount>1) AND
							NOT MAIN.R25.WS[2].DiscreteNode_OK));
		Out_To_ICxx.System_Faults[685]:=Fault_Tmrs[685].Q;
	(*Fault686 - EtherCAT Slave Fault On R26 Water Stand*)
		Fault_Tmrs[686].PT:= No_Timer;
		Fault_Tmrs[686]();
		Fault_Tmrs[686].IN:= (GTAC_CONFIG.Option_Robot_Count>=26)  AND
							(((MAIN.R26.FB_In.Options.WaterStand_Amount>0) AND
							NOT MAIN.R26.WS[1].DiscreteNode_OK) OR
							((MAIN.R26.FB_In.Options.WaterStand_Amount>1) AND
							NOT MAIN.R26.WS[2].DiscreteNode_OK));
		Out_To_ICxx.System_Faults[686]:=Fault_Tmrs[686].Q;
	(*Fault687 - EtherCAT Slave Fault On R27 Water Stand*)
		Fault_Tmrs[687].PT:= No_Timer;
		Fault_Tmrs[687]();
		Fault_Tmrs[687].IN:= (GTAC_CONFIG.Option_Robot_Count>=27)  AND
							(((MAIN.R27.FB_In.Options.WaterStand_Amount>0) AND
							NOT MAIN.R27.WS[1].DiscreteNode_OK) OR
							((MAIN.R27.FB_In.Options.WaterStand_Amount>1) AND
							NOT MAIN.R27.WS[2].DiscreteNode_OK));
		Out_To_ICxx.System_Faults[687]:=Fault_Tmrs[687].Q;
	(*Fault688 - EtherCAT Slave Fault On R28 Water Stand*)
		Fault_Tmrs[688].PT:= No_Timer;
		Fault_Tmrs[688]();
		Fault_Tmrs[688].IN:= (GTAC_CONFIG.Option_Robot_Count>=28)  AND
							(((MAIN.R28.FB_In.Options.WaterStand_Amount>0) AND
							NOT MAIN.R28.WS[1].DiscreteNode_OK) OR
							((MAIN.R28.FB_In.Options.WaterStand_Amount>1) AND
							NOT MAIN.R28.WS[2].DiscreteNode_OK));
		Out_To_ICxx.System_Faults[688]:=Fault_Tmrs[688].Q;
	(*Fault689 - EtherCAT Slave Fault On R29 Water Stand*)
		Fault_Tmrs[689].PT:= No_Timer;
		Fault_Tmrs[689]();
		Fault_Tmrs[689].IN:= (GTAC_CONFIG.Option_Robot_Count>=29)  AND
							(((MAIN.R29.FB_In.Options.WaterStand_Amount>0) AND
							NOT MAIN.R29.WS[1].DiscreteNode_OK) OR
							((MAIN.R29.FB_In.Options.WaterStand_Amount>1) AND
							NOT MAIN.R29.WS[2].DiscreteNode_OK));
		Out_To_ICxx.System_Faults[689]:=Fault_Tmrs[689].Q;
	(*Fault690 - EtherCAT Slave Fault On R30 Water Stand*)
		Fault_Tmrs[690].PT:= No_Timer;
		Fault_Tmrs[690]();
		Fault_Tmrs[690].IN:= (GTAC_CONFIG.Option_Robot_Count>=30)  AND
							(((MAIN.R30.FB_In.Options.WaterStand_Amount>0) AND
							NOT MAIN.R30.WS[1].DiscreteNode_OK) OR
							((MAIN.R30.FB_In.Options.WaterStand_Amount>1) AND
							NOT MAIN.R30.WS[2].DiscreteNode_OK));
		Out_To_ICxx.System_Faults[690]:=Fault_Tmrs[690].Q;


	(*-----------------Rxx EOAT EtherCAT Slave Faulted--------------*)

	(*Fault631 - EtherCAT Slave Fault On EOAT01*)
		Fault_Tmrs[691].PT:= No_Timer;
		Fault_Tmrs[691]();
		Fault_Tmrs[691].IN:= (GTAC_CONFIG.Option_Robot_Count>=1 AND 
							MAIN.R1.FB_In.Options.EOAT_Amount>=1) AND
							NOT EOAT01.DiscreteNode_OK;
		Out_To_ICxx.System_Faults[691]:=Fault_Tmrs[691].Q;
	(*Fault692 - EtherCAT Slave Fault On EOAT02*)
		Fault_Tmrs[692].PT:= No_Timer;
		Fault_Tmrs[692]();
		Fault_Tmrs[692].IN:= (GTAC_CONFIG.Option_Robot_Count>=2 AND 
							MAIN.R2.FB_In.Options.EOAT_Amount>=1) AND
							NOT EOAT02.DiscreteNode_OK;
		Out_To_ICxx.System_Faults[692]:=Fault_Tmrs[692].Q;
	(*Fault693 - EtherCAT Slave Fault On EOAT03*)
		Fault_Tmrs[693].PT:= No_Timer;
		Fault_Tmrs[693]();
		Fault_Tmrs[693].IN:= (GTAC_CONFIG.Option_Robot_Count>=3 AND 
							MAIN.R3.FB_In.Options.EOAT_Amount>=1) AND
							NOT EOAT03.DiscreteNode_OK;
		Out_To_ICxx.System_Faults[693]:=Fault_Tmrs[693].Q;
	(*Fault694 - EtherCAT Slave Fault On EOAT04*)
		Fault_Tmrs[694].PT:= No_Timer;
		Fault_Tmrs[694]();
		Fault_Tmrs[694].IN:= (GTAC_CONFIG.Option_Robot_Count>=4 AND 
							MAIN.R4.FB_In.Options.EOAT_Amount>=1) AND
							NOT EOAT04.DiscreteNode_OK;
		Out_To_ICxx.System_Faults[694]:=Fault_Tmrs[694].Q;
	(*Fault695 - EtherCAT Slave Fault On EOAT05*)
		Fault_Tmrs[695].PT:= No_Timer;
		Fault_Tmrs[695]();
		Fault_Tmrs[695].IN:= (GTAC_CONFIG.Option_Robot_Count>=5 AND 
							MAIN.R5.FB_In.Options.EOAT_Amount>=1) AND
							NOT EOAT05.DiscreteNode_OK;
		Out_To_ICxx.System_Faults[695]:=Fault_Tmrs[695].Q;
	(*Fault696 - EtherCAT Slave Fault In Cabinet06*)
		Fault_Tmrs[696].PT:= No_Timer;
		Fault_Tmrs[696]();
		Fault_Tmrs[696].IN:= (GTAC_CONFIG.Option_Robot_Count>=6 AND 
							MAIN.R6.FB_In.Options.EOAT_Amount>=1) AND
							NOT EOAT06.DiscreteNode_OK;
		Out_To_ICxx.System_Faults[696]:=Fault_Tmrs[696].Q;
	(*Fault697 - EtherCAT Slave Fault On EOAT07*)
		Fault_Tmrs[697].PT:= No_Timer;
		Fault_Tmrs[697]();
		Fault_Tmrs[697].IN:= (GTAC_CONFIG.Option_Robot_Count>=7 AND 
							MAIN.R7.FB_In.Options.EOAT_Amount>=1) AND
							NOT EOAT07.DiscreteNode_OK;
		Out_To_ICxx.System_Faults[697]:=Fault_Tmrs[697].Q;
	(*Fault698 - EtherCAT Slave Fault On EOAT08*)
		Fault_Tmrs[698].PT:= No_Timer;
		Fault_Tmrs[698]();
		Fault_Tmrs[698].IN:= (GTAC_CONFIG.Option_Robot_Count>=8 AND 
							MAIN.R8.FB_In.Options.EOAT_Amount>=1) AND
							NOT EOAT08.DiscreteNode_OK;
		Out_To_ICxx.System_Faults[698]:=Fault_Tmrs[698].Q;
	(*Fault699 - EtherCAT Slave Fault On EOAT09*)
		Fault_Tmrs[699].PT:= No_Timer;
		Fault_Tmrs[699]();
		Fault_Tmrs[699].IN:= (GTAC_CONFIG.Option_Robot_Count>=9 AND 
							MAIN.R9.FB_In.Options.EOAT_Amount>=1) AND
							NOT EOAT09.DiscreteNode_OK;
		Out_To_ICxx.System_Faults[699]:=Fault_Tmrs[699].Q;
	(*Fault700 - EtherCAT Slave Fault On EOAT10*)
		Fault_Tmrs[700].PT:= No_Timer;
		Fault_Tmrs[700]();
		Fault_Tmrs[700].IN:= (GTAC_CONFIG.Option_Robot_Count>=10 AND 
							MAIN.R10.FB_In.Options.EOAT_Amount>=1) AND
							NOT EOAT10.DiscreteNode_OK;
		Out_To_ICxx.System_Faults[700]:=Fault_Tmrs[700].Q;
	(*Fault701 - EtherCAT Slave Fault On EOAT11*)
		Fault_Tmrs[701].PT:= No_Timer;
		Fault_Tmrs[701]();
		Fault_Tmrs[701].IN:= FALSE;
		Out_To_ICxx.System_Faults[701]:=Fault_Tmrs[701].Q;
	(*Fault702 - EtherCAT Slave Fault On EOAT12*)
		Fault_Tmrs[702].PT:= No_Timer;
		Fault_Tmrs[702]();
		Fault_Tmrs[702].IN:= FALSE;
		Out_To_ICxx.System_Faults[702]:=Fault_Tmrs[702].Q;
	(*Fault703 - EtherCAT Slave Fault On EOAT13*)
		Fault_Tmrs[703].PT:= No_Timer;
		Fault_Tmrs[703]();
		Fault_Tmrs[703].IN:= FALSE;
		Out_To_ICxx.System_Faults[703]:=Fault_Tmrs[703].Q;
	(*Fault704 - EtherCAT Slave Fault On EOAT14*)
		Fault_Tmrs[704].PT:= No_Timer;
		Fault_Tmrs[704]();
		Fault_Tmrs[704].IN:= FALSE;
		Out_To_ICxx.System_Faults[704]:=Fault_Tmrs[704].Q;
	(*Fault705 - EtherCAT Slave Fault On EOAT15*)
		Fault_Tmrs[705].PT:= No_Timer;
		Fault_Tmrs[705]();
		Fault_Tmrs[705].IN:= FALSE;
		Out_To_ICxx.System_Faults[705]:=Fault_Tmrs[705].Q;
	(*Fault706 - EtherCAT Slave Fault On EOAT16*)
		Fault_Tmrs[706].PT:= No_Timer;
		Fault_Tmrs[706]();
		Fault_Tmrs[706].IN:= FALSE;
		Out_To_ICxx.System_Faults[706]:=Fault_Tmrs[706].Q;
	(*Fault707 - EtherCAT Slave Fault On EOAT17*)
		Fault_Tmrs[707].PT:= No_Timer;
		Fault_Tmrs[707]();
		Fault_Tmrs[707].IN:= FALSE;
		Out_To_ICxx.System_Faults[707]:=Fault_Tmrs[707].Q;
	(*Fault708 - EtherCAT Slave Fault On EOAT18*)
		Fault_Tmrs[708].PT:= No_Timer;
		Fault_Tmrs[708]();
		Fault_Tmrs[708].IN:= FALSE;
		Out_To_ICxx.System_Faults[708]:=Fault_Tmrs[708].Q;
	(*Fault709 - EtherCAT Slave Fault On EOAT19*)
		Fault_Tmrs[709].PT:= No_Timer;
		Fault_Tmrs[709]();
		Fault_Tmrs[709].IN:= FALSE;
		Out_To_ICxx.System_Faults[709]:=Fault_Tmrs[709].Q;
	(*Fault710 - EtherCAT Slave Fault On EOAT20*)
		Fault_Tmrs[710].PT:= No_Timer;
		Fault_Tmrs[710]();
		Fault_Tmrs[710].IN:= FALSE;
		Out_To_ICxx.System_Faults[710]:=Fault_Tmrs[710].Q;
	(*Fault711 - EtherCAT Slave Fault On EOAT21*)
		Fault_Tmrs[711].PT:= No_Timer;
		Fault_Tmrs[711]();
		Fault_Tmrs[711].IN:= FALSE;
		Out_To_ICxx.System_Faults[711]:=Fault_Tmrs[711].Q;
	(*Fault712 - EtherCAT Slave Fault On EOAT22*)
		Fault_Tmrs[712].PT:= No_Timer;
		Fault_Tmrs[712]();
		Fault_Tmrs[712].IN:= FALSE;
		Out_To_ICxx.System_Faults[712]:=Fault_Tmrs[712].Q;
	(*Fault713 - EtherCAT Slave Fault On EOAT23*)
		Fault_Tmrs[713].PT:= No_Timer;
		Fault_Tmrs[713]();
		Fault_Tmrs[713].IN:= FALSE;
		Out_To_ICxx.System_Faults[713]:=Fault_Tmrs[713].Q;
	(*Fault714 - EtherCAT Slave Fault On EOAT24*)
		Fault_Tmrs[714].PT:= No_Timer;
		Fault_Tmrs[714]();
		Fault_Tmrs[714].IN:= FALSE;
		Out_To_ICxx.System_Faults[714]:=Fault_Tmrs[714].Q;
	(*Fault715 - EtherCAT Slave Fault On EOAT25*)
		Fault_Tmrs[715].PT:= No_Timer;
		Fault_Tmrs[715]();
		Fault_Tmrs[715].IN:= FALSE;
		Out_To_ICxx.System_Faults[715]:=Fault_Tmrs[715].Q;
	(*Fault716 - EtherCAT Slave Fault On EOAT26*)
		Fault_Tmrs[716].PT:= No_Timer;
		Fault_Tmrs[716]();
		Fault_Tmrs[716].IN:= FALSE;
		Out_To_ICxx.System_Faults[716]:=Fault_Tmrs[716].Q;
	(*Fault717 - EtherCAT Slave Fault On EOAT27*)
		Fault_Tmrs[717].PT:= No_Timer;
		Fault_Tmrs[717]();
		Fault_Tmrs[717].IN:= FALSE;
		Out_To_ICxx.System_Faults[717]:=Fault_Tmrs[717].Q;
	(*Fault718 - EtherCAT Slave Fault On EOAT28*)
		Fault_Tmrs[718].PT:= No_Timer;
		Fault_Tmrs[718]();
		Fault_Tmrs[718].IN:= FALSE;
		Out_To_ICxx.System_Faults[718]:=Fault_Tmrs[718].Q;
	(*Fault719 - EtherCAT Slave Fault On EOAT29*)
		Fault_Tmrs[719].PT:= No_Timer;
		Fault_Tmrs[719]();
		Fault_Tmrs[719].IN:=FALSE;
		Out_To_ICxx.System_Faults[719]:=Fault_Tmrs[719].Q;
	(*Fault720 - EtherCAT Slave Fault On EOAT30*)
		Fault_Tmrs[720].PT:= No_Timer;
		Fault_Tmrs[720]();
		Fault_Tmrs[720].IN:= FALSE;
		Out_To_ICxx.System_Faults[720]:=Fault_Tmrs[720].Q;



	(*-----------------SD EtherCAT Slave Faults--------------*)
	(*Fault721 - EtherCAT Slave Fault in SD1 (Drive or integrated safety card if appl.)*)
		Fault_Tmrs[721].PT:= No_Timer;
		Fault_Tmrs[721]();
		Fault_Tmrs[721].IN:= (GTAC_CONFIG.Option_SD_Count>=1) AND
							NOT Servo_Motion.SD[1].DiscreteNode_OK;
		Out_To_ICxx.System_Faults[721]:=Fault_Tmrs[721].Q;
	(*Fault722 - EtherCAT Slave Fault in SD2 (Drive or integrated safety card if appl.)*)
		Fault_Tmrs[722].PT:= No_Timer;
		Fault_Tmrs[722]();
		Fault_Tmrs[722].IN:= (GTAC_CONFIG.Option_SD_Count>=2) AND
							NOT Servo_Motion.SD[2].DiscreteNode_OK;
		Out_To_ICxx.System_Faults[722]:=Fault_Tmrs[722].Q;
	(*Fault723 - EtherCAT Slave Fault in SD3 (Drive or integrated safety card if appl.)*)
		Fault_Tmrs[723].PT:= No_Timer;
		Fault_Tmrs[723]();
		Fault_Tmrs[723].IN:= (GTAC_CONFIG.Option_SD_Count>=3) AND
							NOT Servo_Motion.SD[3].DiscreteNode_OK;
		Out_To_ICxx.System_Faults[723]:=Fault_Tmrs[723].Q;
	(*Fault724 - EtherCAT Slave Fault in SD4 (Drive or integrated safety card if appl.)*)
		Fault_Tmrs[724].PT:= No_Timer;
		Fault_Tmrs[724]();
		Fault_Tmrs[724].IN:= (GTAC_CONFIG.Option_SD_Count>=4) AND
							NOT Servo_Motion.SD[4].DiscreteNode_OK;
		Out_To_ICxx.System_Faults[724]:=Fault_Tmrs[724].Q;
	(*Fault725 - EtherCAT Slave Fault in SD5 (Drive or integrated safety card if appl.)*)
		Fault_Tmrs[725].PT:= No_Timer;
		Fault_Tmrs[725]();
		Fault_Tmrs[725].IN:= (GTAC_CONFIG.Option_SD_Count>=5) AND
							NOT Servo_Motion.SD[5].DiscreteNode_OK;
		Out_To_ICxx.System_Faults[725]:=Fault_Tmrs[725].Q;
	(*Fault726 - EtherCAT Slave Fault in SD6 (Drive or integrated safety card if appl.)*)
		Fault_Tmrs[726].PT:= No_Timer;
		Fault_Tmrs[726]();
		Fault_Tmrs[726].IN:= (GTAC_CONFIG.Option_SD_Count>=6) AND
							NOT Servo_Motion.SD[6].DiscreteNode_OK;
		Out_To_ICxx.System_Faults[726]:=Fault_Tmrs[726].Q;
	(*Fault727 - EtherCAT Slave Fault in SD7 (Drive or integrated safety card if appl.)*)
		Fault_Tmrs[727].PT:= No_Timer;
		Fault_Tmrs[727]();
		Fault_Tmrs[727].IN:= (GTAC_CONFIG.Option_SD_Count>=7) AND
							NOT Servo_Motion.SD[7].DiscreteNode_OK;
		Out_To_ICxx.System_Faults[727]:=Fault_Tmrs[727].Q;
	(*Fault728 - EtherCAT Slave Fault in SD8 (Drive or integrated safety card if appl.)*)
		Fault_Tmrs[728].PT:= No_Timer;
		Fault_Tmrs[728]();
		Fault_Tmrs[728].IN:= (GTAC_CONFIG.Option_SD_Count>=8) AND
							NOT Servo_Motion.SD[8].DiscreteNode_OK;
		Out_To_ICxx.System_Faults[728]:=Fault_Tmrs[728].Q;
	(*Fault729 - EtherCAT Slave Fault in SD9 (Drive or integrated safety card if appl.)*)
		Fault_Tmrs[729].PT:= No_Timer;
		Fault_Tmrs[729]();
		Fault_Tmrs[729].IN:= (GTAC_CONFIG.Option_SD_Count>=9) AND
							NOT Servo_Motion.SD[9].DiscreteNode_OK;
		Out_To_ICxx.System_Faults[729]:=Fault_Tmrs[729].Q;
	(*Fault730 - EtherCAT Slave Fault in SD10 (Drive or integrated safety card if appl.)*)
		Fault_Tmrs[730].PT:= No_Timer;
		Fault_Tmrs[730]();
		Fault_Tmrs[730].IN:= (GTAC_CONFIG.Option_SD_Count>=10) AND
							NOT Servo_Motion.SD[10].DiscreteNode_OK;
		Out_To_ICxx.System_Faults[730]:=Fault_Tmrs[730].Q;
	(*Fault731 - EtherCAT Slave Fault in SD11 (Drive or integrated safety card if appl.)*)
		Fault_Tmrs[731].PT:= No_Timer;
		Fault_Tmrs[731]();
		Fault_Tmrs[731].IN:= (GTAC_CONFIG.Option_SD_Count>=11) AND
							NOT Servo_Motion.SD[11].DiscreteNode_OK;
		Out_To_ICxx.System_Faults[731]:=Fault_Tmrs[731].Q;
	(*Fault732 - EtherCAT Slave Fault in SD12 (Drive or integrated safety card if appl.)*)
		Fault_Tmrs[732].PT:= No_Timer;
		Fault_Tmrs[732]();
		Fault_Tmrs[732].IN:= (GTAC_CONFIG.Option_SD_Count>=12) AND
							NOT Servo_Motion.SD[12].DiscreteNode_OK;
		Out_To_ICxx.System_Faults[732]:=Fault_Tmrs[732].Q;
	(*Fault733 - EtherCAT Slave Fault in SD13 (Drive or integrated safety card if appl.)*)
		Fault_Tmrs[733].PT:= No_Timer;
		Fault_Tmrs[733]();
		Fault_Tmrs[733].IN:= (GTAC_CONFIG.Option_SD_Count>=13) AND
							NOT Servo_Motion.SD[13].DiscreteNode_OK;
		Out_To_ICxx.System_Faults[733]:=Fault_Tmrs[733].Q;
	(*Fault734 - EtherCAT Slave Fault in SD14 (Drive or integrated safety card if appl.)*)
		Fault_Tmrs[734].PT:= No_Timer;
		Fault_Tmrs[734]();
		Fault_Tmrs[734].IN:= (GTAC_CONFIG.Option_SD_Count>=14) AND
							NOT Servo_Motion.SD[14].DiscreteNode_OK;
		Out_To_ICxx.System_Faults[734]:=Fault_Tmrs[734].Q;
	(*Fault735 - EtherCAT Slave Fault in SD15 (Drive or integrated safety card if appl.)*)
		Fault_Tmrs[735].PT:= No_Timer;
		Fault_Tmrs[735]();
		Fault_Tmrs[735].IN:= (GTAC_CONFIG.Option_SD_Count>=15) AND
							NOT Servo_Motion.SD[15].DiscreteNode_OK;
		Out_To_ICxx.System_Faults[735]:=Fault_Tmrs[735].Q;
	(*Fault736 - EtherCAT Slave Fault in SD16 (Drive or integrated safety card if appl.)*)
		Fault_Tmrs[736].PT:= No_Timer;
		Fault_Tmrs[736]();
		Fault_Tmrs[736].IN:= (GTAC_CONFIG.Option_SD_Count>=16) AND
							NOT Servo_Motion.SD[16].DiscreteNode_OK;
		Out_To_ICxx.System_Faults[736]:=Fault_Tmrs[736].Q;
	(*Fault737 - EtherCAT Slave Fault in SD17 (Drive or integrated safety card if appl.)*)
		Fault_Tmrs[737].PT:= No_Timer;
		Fault_Tmrs[737]();
		Fault_Tmrs[737].IN:= (GTAC_CONFIG.Option_SD_Count>=17) AND
							NOT Servo_Motion.SD[17].DiscreteNode_OK;
		Out_To_ICxx.System_Faults[737]:=Fault_Tmrs[737].Q;
	(*Fault738 - EtherCAT Slave Fault in SD18 (Drive or integrated safety card if appl.)*)
		Fault_Tmrs[738].PT:= No_Timer;
		Fault_Tmrs[738]();
		Fault_Tmrs[738].IN:= (GTAC_CONFIG.Option_SD_Count>=18) AND
							NOT Servo_Motion.SD[18].DiscreteNode_OK;
		Out_To_ICxx.System_Faults[738]:=Fault_Tmrs[738].Q;
	(*Fault739 - EtherCAT Slave Fault in SD19 (Drive or integrated safety card if appl.)*)
		Fault_Tmrs[739].PT:= No_Timer;
		Fault_Tmrs[739]();
		Fault_Tmrs[739].IN:= (GTAC_CONFIG.Option_SD_Count>=19) AND
							NOT Servo_Motion.SD[19].DiscreteNode_OK;
		Out_To_ICxx.System_Faults[739]:=Fault_Tmrs[739].Q;
	(*Fault740 - EtherCAT Slave Fault in SD20 (Drive or integrated safety card if appl.)*)
		Fault_Tmrs[740].PT:= No_Timer;
		Fault_Tmrs[740]();
		Fault_Tmrs[740].IN:= (GTAC_CONFIG.Option_SD_Count>=20) AND
							NOT Servo_Motion.SD[20].DiscreteNode_OK;
		Out_To_ICxx.System_Faults[740]:=Fault_Tmrs[740].Q;
	(*Fault741 - EtherCAT Slave Fault in SD21 (Drive or integrated safety card if appl.)*)
		Fault_Tmrs[741].PT:= No_Timer;
		Fault_Tmrs[741]();
		Fault_Tmrs[741].IN:= (GTAC_CONFIG.Option_SD_Count>=21) AND
							NOT Servo_Motion.SD[21].DiscreteNode_OK;
		Out_To_ICxx.System_Faults[741]:=Fault_Tmrs[741].Q;
	(*Fault742 - EtherCAT Slave Fault in SD22 (Drive or integrated safety card if appl.)*)
		Fault_Tmrs[742].PT:= No_Timer;
		Fault_Tmrs[742]();
		Fault_Tmrs[742].IN:= (GTAC_CONFIG.Option_SD_Count>=22) AND
							NOT Servo_Motion.SD[22].DiscreteNode_OK;
		Out_To_ICxx.System_Faults[742]:=Fault_Tmrs[742].Q;
	(*Fault743 - EtherCAT Slave Fault in SD23 (Drive or integrated safety card if appl.)*)
		Fault_Tmrs[743].PT:= No_Timer;
		Fault_Tmrs[743]();
		Fault_Tmrs[743].IN:= (GTAC_CONFIG.Option_SD_Count>=23) AND
							NOT Servo_Motion.SD[23].DiscreteNode_OK;
		Out_To_ICxx.System_Faults[743]:=Fault_Tmrs[743].Q;
	(*Fault744 - EtherCAT Slave Fault in SD24 (Drive or integrated safety card if appl.)*)
		Fault_Tmrs[744].PT:= No_Timer;
		Fault_Tmrs[744]();
		Fault_Tmrs[744].IN:= (GTAC_CONFIG.Option_SD_Count>=24) AND
							NOT Servo_Motion.SD[24].DiscreteNode_OK;
		Out_To_ICxx.System_Faults[744]:=Fault_Tmrs[744].Q;
	(*Fault745 - EtherCAT Slave Fault in SD25 (Drive or integrated safety card if appl.)*)
		Fault_Tmrs[745].PT:= No_Timer;
		Fault_Tmrs[745]();
		Fault_Tmrs[745].IN:= (GTAC_CONFIG.Option_SD_Count>=25) AND
							NOT Servo_Motion.SD[25].DiscreteNode_OK;
		Out_To_ICxx.System_Faults[745]:=Fault_Tmrs[745].Q;
	(*Fault746 - EtherCAT Slave Fault in SD26 (Drive or integrated safety card if appl.)*)
		Fault_Tmrs[746].PT:= No_Timer;
		Fault_Tmrs[746]();
		Fault_Tmrs[746].IN:= (GTAC_CONFIG.Option_SD_Count>=26) AND
							NOT Servo_Motion.SD[26].DiscreteNode_OK;
		Out_To_ICxx.System_Faults[746]:=Fault_Tmrs[746].Q;
	(*Fault747 - EtherCAT Slave Fault in SD27 (Drive or integrated safety card if appl.)*)
		Fault_Tmrs[747].PT:= No_Timer;
		Fault_Tmrs[747]();
		Fault_Tmrs[747].IN:= (GTAC_CONFIG.Option_SD_Count>=27) AND
							NOT Servo_Motion.SD[27].DiscreteNode_OK;
		Out_To_ICxx.System_Faults[747]:=Fault_Tmrs[747].Q;
	(*Fault748 - EtherCAT Slave Fault in SD28 (Drive or integrated safety card if appl.)*)
		Fault_Tmrs[748].PT:= No_Timer;
		Fault_Tmrs[748]();
		Fault_Tmrs[748].IN:= (GTAC_CONFIG.Option_SD_Count>=28) AND
							NOT Servo_Motion.SD[28].DiscreteNode_OK;
		Out_To_ICxx.System_Faults[748]:=Fault_Tmrs[748].Q;
	(*Fault749 - EtherCAT Slave Fault in SD29 (Drive or integrated safety card if appl.)*)
		Fault_Tmrs[749].PT:= No_Timer;
		Fault_Tmrs[749]();
		Fault_Tmrs[749].IN:= (GTAC_CONFIG.Option_SD_Count>=29) AND
							NOT Servo_Motion.SD[29].DiscreteNode_OK;
		Out_To_ICxx.System_Faults[749]:=Fault_Tmrs[749].Q;
	(*Fault750 - EtherCAT Slave Fault in SD30 (Drive or integrated safety card if appl.)*)
		Fault_Tmrs[750].PT:= No_Timer;
		Fault_Tmrs[750]();
		Fault_Tmrs[750].IN:= (GTAC_CONFIG.Option_SD_Count>=30) AND
							NOT Servo_Motion.SD[30].DiscreteNode_OK;
		Out_To_ICxx.System_Faults[750]:=Fault_Tmrs[750].Q;
		
	(*--------- VFD EtherCAT Slave Faults ----------------*)
	(*Fault751 - EtherCAT Slave Fault in VFD01*)
		Fault_Tmrs[751].PT:= No_Timer;
		Fault_Tmrs[751]();
		Fault_Tmrs[751].IN:= (GTAC_CONFIG.Option_VFD_Count>=1) AND
							NOT MAIN.VFD01.DiscreteNode_OK;
		Out_To_ICxx.System_Faults[751]:=Fault_Tmrs[751].Q;
	(*Fault752 - EtherCAT Slave Fault in VFD02*)
		Fault_Tmrs[752].PT:= No_Timer;
		Fault_Tmrs[752]();
		Fault_Tmrs[752].IN:= (GTAC_CONFIG.Option_VFD_Count>=2) AND
							NOT MAIN.VFD02.DiscreteNode_OK;
		Out_To_ICxx.System_Faults[752]:=Fault_Tmrs[752].Q;
	(*Fault753 - EtherCAT Slave Fault in VFD03*)
		Fault_Tmrs[753].PT:= No_Timer;
		Fault_Tmrs[753]();
		Fault_Tmrs[753].IN:= (GTAC_CONFIG.Option_VFD_Count>=3) AND
							NOT MAIN.VFD03.DiscreteNode_OK;
		Out_To_ICxx.System_Faults[753]:=Fault_Tmrs[753].Q;
	(*Fault754 - EtherCAT Slave Fault in VFD04*)
		Fault_Tmrs[754].PT:= No_Timer;
		Fault_Tmrs[754]();
		Fault_Tmrs[754].IN:= (GTAC_CONFIG.Option_VFD_Count>=4) AND
							NOT MAIN.VFD04.DiscreteNode_OK;
		Out_To_ICxx.System_Faults[754]:=Fault_Tmrs[754].Q;
	(*Fault755 - EtherCAT Slave Fault in VFD05*)
		Fault_Tmrs[755].PT:= No_Timer;
		Fault_Tmrs[755]();
		Fault_Tmrs[755].IN:= (GTAC_CONFIG.Option_VFD_Count>=5) AND
							NOT MAIN.VFD05.DiscreteNode_OK;
		Out_To_ICxx.System_Faults[755]:=Fault_Tmrs[755].Q;
			
	
	(*----------------- LSR EtherCAT Slave Faults --------------*)
	
	(*Fault756 - EtherCAT Slave Fault in LSR01*)
		Fault_Tmrs[756].PT:= No_Timer;
		Fault_Tmrs[756]();
		Fault_Tmrs[756].IN:= NOT Main.Laser01.DiscreteNode_OK AND FALSE;
		Out_To_ICxx.System_Faults[756]:=Fault_Tmrs[756].Q;

	(*Fault757 - EtherCAT Slave Fault in LSR02*)
		Fault_Tmrs[757].PT:= No_Timer;
		Fault_Tmrs[757]();
		Fault_Tmrs[757].IN:= FALSE;
		Out_To_ICxx.System_Faults[757]:=Fault_Tmrs[757].Q;
	
	(*-------------------------------------------------------------- Network/Cable Disconnect Faults --------------------------------------------------------*)
	
	(*Fault761 - Ecat Master in IPC to IC01 Cable disconnected*)
		Fault_Tmrs[761].PT:=No_Timer;
		Fault_Tmrs[761]();
		Fault_Tmrs[761].IN:= (GTAC_CONFIG.Option_IC_Count>=1) AND
							MAIN.IC01.EK1100_NotPresent;
		Out_To_ICxx.System_Faults[761]:=Fault_Tmrs[761].Q;

	(*Fault762 - IC01 EK1100 Out Port Cable disconnected*)
		Fault_Tmrs[762].PT:=No_Timer;
		Fault_Tmrs[762]();
		Fault_Tmrs[762].IN:= (GTAC_CONFIG.Option_IC_Count>=1) AND
							MAIN.IC01.EK1100_PortC_MissingLink;
		Out_To_ICxx.System_Faults[762]:=Fault_Tmrs[762].Q;
	(*Fault763 - IC01 EK1122 OP1 Cable disconnected (X1)*)
		Fault_Tmrs[763].PT:=No_Timer;
		Fault_Tmrs[763]();
		Fault_Tmrs[763].IN:= (GTAC_CONFIG.Option_IC_Count>=1) AND
							MAIN.IC01.EK1122_PortD_MissingLink;
		Out_To_ICxx.System_Faults[763]:=Fault_Tmrs[763].Q;
	(*Fault764 - IC01 EK1122 OP2 Cable disconnected (X2)*)
		Fault_Tmrs[764].PT:=No_Timer;
		Fault_Tmrs[764]();
		Fault_Tmrs[764].IN:= (GTAC_CONFIG.Option_IC_Count>=1) AND
							MAIN.IC01.EK1122_PortB_MissingLink;
		Out_To_ICxx.System_Faults[764]:=Fault_Tmrs[764].Q;

	(*Fault766 - IC02 EK1100 Out Port Cable disconnected*)
		Fault_Tmrs[766].PT:=No_Timer;
		Fault_Tmrs[766]();
		Fault_Tmrs[766].IN:= (GTAC_CONFIG.Option_IC_Count>=2) AND
							MAIN.IC02.EK1100_PortC_MissingLink;
		Out_To_ICxx.System_Faults[766]:=Fault_Tmrs[766].Q;
	(*Fault767 - IC02 EK1122 OP1 Cable disconnected (X1)*)
		Fault_Tmrs[767].PT:=No_Timer;
		Fault_Tmrs[767]();
		Fault_Tmrs[767].IN:= (GTAC_CONFIG.Option_IC_Count>=2) AND
							MAIN.IC02.EK1122_PortD_MissingLink;
		Out_To_ICxx.System_Faults[767]:=Fault_Tmrs[767].Q;
	(*Fault768 - IC02 EK1122 OP2 Cable disconnected (X2)*)
		Fault_Tmrs[768].PT:=No_Timer;
		Fault_Tmrs[768]();
		Fault_Tmrs[768].IN:= (GTAC_CONFIG.Option_IC_Count>=2) AND
							MAIN.IC02.EK1122_PortB_MissingLink;
		Out_To_ICxx.System_Faults[768]:=Fault_Tmrs[768].Q;

	(*Fault770 - IC03 EK1100 Out Port Cable disconnected*)
		Fault_Tmrs[770].PT:=No_Timer;
		Fault_Tmrs[770]();
		Fault_Tmrs[770].IN:= (GTAC_CONFIG.Option_IC_Count>=3) AND
							MAIN.IC03.EK1100_PortC_MissingLink;
		Out_To_ICxx.System_Faults[770]:=Fault_Tmrs[770].Q;
	(*Fault771 - IC03 EK1122 OP1 Cable disconnected (X1)*)
		Fault_Tmrs[771].PT:=No_Timer;
		Fault_Tmrs[771]();
		Fault_Tmrs[771].IN:= (GTAC_CONFIG.Option_IC_Count>=3) AND
							MAIN.IC03.EK1122_PortD_MissingLink;
		Out_To_ICxx.System_Faults[771]:=Fault_Tmrs[771].Q;
	(*Fault772 - IC03 EK1122 OP2 Cable disconnected (X2)*)
		Fault_Tmrs[772].PT:=No_Timer;
		Fault_Tmrs[772]();
		Fault_Tmrs[772].IN:= (GTAC_CONFIG.Option_IC_Count>=3) AND
							MAIN.IC03.EK1122_PortB_MissingLink;
		Out_To_ICxx.System_Faults[772]:=Fault_Tmrs[772].Q;

	(*Fault774 - IC04 EK1100 Out Port Cable disconnected*)
		Fault_Tmrs[774].PT:=No_Timer;
		Fault_Tmrs[774]();
		Fault_Tmrs[774].IN:= (GTAC_CONFIG.Option_IC_Count>=4) AND
							MAIN.IC04.EK1100_PortC_MissingLink;
		Out_To_ICxx.System_Faults[774]:=Fault_Tmrs[774].Q;
	(*Fault775 - IC04 EK1122 OP1 Cable disconnected (X1)*)
		Fault_Tmrs[775].PT:=No_Timer;
		Fault_Tmrs[775]();
		Fault_Tmrs[775].IN:= (GTAC_CONFIG.Option_IC_Count>=4) AND
							MAIN.IC04.EK1122_PortD_MissingLink;
		Out_To_ICxx.System_Faults[775]:=Fault_Tmrs[775].Q;
	(*Fault776 - IC04 EK1122 OP2 Cable disconnected (X2)*)
		Fault_Tmrs[776].PT:=No_Timer;
		Fault_Tmrs[776]();
		Fault_Tmrs[776].IN:= (GTAC_CONFIG.Option_IC_Count>=4) AND
							MAIN.IC04.EK1122_PortB_MissingLink;
		Out_To_ICxx.System_Faults[776]:=Fault_Tmrs[776].Q;

	(*Fault778 - IC05 EK1100 Out Port Cable disconnected*)
		Fault_Tmrs[778].PT:=No_Timer;
		Fault_Tmrs[778]();
		Fault_Tmrs[778].IN:= (GTAC_CONFIG.Option_IC_Count>=5) AND
							MAIN.IC05.EK1100_PortC_MissingLink;
		Out_To_ICxx.System_Faults[778]:=Fault_Tmrs[778].Q;
	(*Fault779 - IC05 EK1122 OP1 Cable disconnected (X1)*)
		Fault_Tmrs[779].PT:=No_Timer;
		Fault_Tmrs[779]();
		Fault_Tmrs[779].IN:= (GTAC_CONFIG.Option_IC_Count>=5) AND
							MAIN.IC05.EK1122_PortD_MissingLink;
		Out_To_ICxx.System_Faults[779]:=Fault_Tmrs[779].Q;
	(*Fault780 - IC05 EK1122 OP2 Cable disconnected (X2)*)
		Fault_Tmrs[780].PT:=No_Timer;
		Fault_Tmrs[780]();
		Fault_Tmrs[780].IN:= (GTAC_CONFIG.Option_IC_Count>=5) AND
							MAIN.IC05.EK1122_PortB_MissingLink;
		Out_To_ICxx.System_Faults[780]:=Fault_Tmrs[780].Q;

	(*Fault782 - IC06 EK1100 Out Port Cable disconnected*)
		Fault_Tmrs[782].PT:=No_Timer;
		Fault_Tmrs[782]();
		Fault_Tmrs[782].IN:= (GTAC_CONFIG.Option_IC_Count>=6) AND
							MAIN.IC06.EK1100_PortC_MissingLink;
		Out_To_ICxx.System_Faults[782]:=Fault_Tmrs[782].Q;
	(*Fault783 - IC06 EK1122 OP1 Cable disconnected (X1)*)
		Fault_Tmrs[783].PT:=No_Timer;
		Fault_Tmrs[783]();
		Fault_Tmrs[783].IN:= (GTAC_CONFIG.Option_IC_Count>=6) AND
							MAIN.IC06.EK1122_PortD_MissingLink;
		Out_To_ICxx.System_Faults[783]:=Fault_Tmrs[783].Q;
	(*Fault784 - IC06 EK1122 OP2 Cable disconnected (X2)*)
		Fault_Tmrs[784].PT:=No_Timer;
		Fault_Tmrs[784]();
		Fault_Tmrs[784].IN:= (GTAC_CONFIG.Option_IC_Count>=6) AND
							MAIN.IC06.EK1122_PortB_MissingLink;
		Out_To_ICxx.System_Faults[784]:=Fault_Tmrs[784].Q;

	(*Fault786 - IC07 EK1100 Out Port Cable disconnected*)
		Fault_Tmrs[786].PT:=No_Timer;
		Fault_Tmrs[786]();
		Fault_Tmrs[786].IN:= (GTAC_CONFIG.Option_IC_Count>=7) AND
							MAIN.IC07.EK1100_PortC_MissingLink;
		Out_To_ICxx.System_Faults[786]:=Fault_Tmrs[786].Q;
	(*Fault787 - IC07 EK1122 OP1 Cable disconnected (X1)*)
		Fault_Tmrs[787].PT:=No_Timer;
		Fault_Tmrs[787]();
		Fault_Tmrs[787].IN:= (GTAC_CONFIG.Option_IC_Count>=7) AND
							MAIN.IC07.EK1122_PortD_MissingLink;
		Out_To_ICxx.System_Faults[787]:=Fault_Tmrs[787].Q;
	(*Fault788 - IC07 EK1122 OP2 Cable disconnected (X2)*)
		Fault_Tmrs[788].PT:=No_Timer;
		Fault_Tmrs[788]();
		Fault_Tmrs[788].IN:= (GTAC_CONFIG.Option_IC_Count>=7) AND
						MAIN.IC07.EK1122_PortB_MissingLink;
		Out_To_ICxx.System_Faults[788]:=Fault_Tmrs[788].Q;

	(*Fault790 - IC08 EK1100 Out Port Cable disconnected*)
		Fault_Tmrs[790].PT:=No_Timer;
		Fault_Tmrs[790]();
		Fault_Tmrs[790].IN:= (GTAC_CONFIG.Option_IC_Count>=8) AND
							MAIN.IC08.EK1100_PortC_MissingLink;
		Out_To_ICxx.System_Faults[790]:=Fault_Tmrs[790].Q;
	(*Fault791 - IC08 EK1122 OP1 Cable disconnected (X1)*)
		Fault_Tmrs[791].PT:=No_Timer;
		Fault_Tmrs[791]();
		Fault_Tmrs[791].IN:= (GTAC_CONFIG.Option_IC_Count>=8) AND
							MAIN.IC08.EK1122_PortD_MissingLink;
		Out_To_ICxx.System_Faults[791]:=Fault_Tmrs[791].Q;
	(*Fault792 - IC08 EK1122 OP2 Cable disconnected (X2)*)
		Fault_Tmrs[792].PT:=No_Timer;
		Fault_Tmrs[792]();
		Fault_Tmrs[792].IN:= (GTAC_CONFIG.Option_IC_Count>=8) AND
							MAIN.IC08.EK1122_PortB_MissingLink;
		Out_To_ICxx.System_Faults[792]:=Fault_Tmrs[792].Q;

	(*Internal Fixtures*)
	(*Faults 794 -805 reserved for internal tool disconnects*)
	(*DEBUG add as required*)

	(*Robots*)
	(*-----Out Port Cable-------*)
	(*Fault811 - R01 EK1100 Out Port Cabe disconnected*)
		Fault_Tmrs[811].PT:=No_Timer;
		Fault_Tmrs[811]();
		Fault_Tmrs[811].IN:= (GTAC_CONFIG.Option_Robot_Count>=1) AND
							MAIN.R1.EL6695_PortC_MissingLink;
		Out_To_ICxx.System_Faults[811]:=Fault_Tmrs[811].Q;
	(*Fault812 - R02 EK1100 Out Port Cabe disconnected*)
		Fault_Tmrs[812].PT:=No_Timer;
		Fault_Tmrs[812]();
		Fault_Tmrs[812].IN:= (GTAC_CONFIG.Option_Robot_Count>=2) AND
							MAIN.R2.EL6695_PortC_MissingLink;
		Out_To_ICxx.System_Faults[812]:=Fault_Tmrs[812].Q;
	(*Fault813 - R03 EK1100 Out Port Cabe disconnected*)
		Fault_Tmrs[813].PT:=No_Timer;
		Fault_Tmrs[813]();
		Fault_Tmrs[813].IN:= (GTAC_CONFIG.Option_Robot_Count>=3) AND
							MAIN.R3.EL6695_PortC_MissingLink;
		Out_To_ICxx.System_Faults[813]:=Fault_Tmrs[813].Q;
	(*Fault814 - R04 EK1100 Out Port Cabe disconnected*)
		Fault_Tmrs[814].PT:=No_Timer;
		Fault_Tmrs[814]();
		Fault_Tmrs[814].IN:= (GTAC_CONFIG.Option_Robot_Count>=4) AND
							MAIN.R4.EL6695_PortC_MissingLink;
		Out_To_ICxx.System_Faults[814]:=Fault_Tmrs[814].Q;
	(*Fault815 - R05 EK1100 Out Port Cabe disconnected*)
		Fault_Tmrs[815].PT:=No_Timer;
		Fault_Tmrs[815]();
		Fault_Tmrs[815].IN:= (GTAC_CONFIG.Option_Robot_Count>=5) AND
							MAIN.R5.EL6695_PortC_MissingLink;
		Out_To_ICxx.System_Faults[815]:=Fault_Tmrs[815].Q;
	(*Fault816 - R06 EK1100 Out Port Cabe disconnected*)
		Fault_Tmrs[816].PT:=No_Timer;
		Fault_Tmrs[816]();
		Fault_Tmrs[816].IN:= (GTAC_CONFIG.Option_Robot_Count>=6) AND
							MAIN.R6.EL6695_PortC_MissingLink;
		Out_To_ICxx.System_Faults[816]:=Fault_Tmrs[816].Q;
	(*Fault817 - R07 EK1100 Out Port Cabe disconnected*)
		Fault_Tmrs[817].PT:=No_Timer;
		Fault_Tmrs[817]();
		Fault_Tmrs[817].IN:= (GTAC_CONFIG.Option_Robot_Count>=7) AND
							MAIN.R7.EL6695_PortC_MissingLink;
		Out_To_ICxx.System_Faults[817]:=Fault_Tmrs[817].Q;
	(*Fault818 - R08 EK1100 Out Port Cabe disconnected*)
		Fault_Tmrs[818].PT:=No_Timer;
		Fault_Tmrs[818]();
		Fault_Tmrs[818].IN:= (GTAC_CONFIG.Option_Robot_Count>=8) AND
							MAIN.R8.EL6695_PortC_MissingLink;
		Out_To_ICxx.System_Faults[818]:=Fault_Tmrs[818].Q;
	(*Fault819 - R09 EK1100 Out Port Cabe disconnected*)
		Fault_Tmrs[819].PT:=No_Timer;
		Fault_Tmrs[819]();
		Fault_Tmrs[819].IN:= (GTAC_CONFIG.Option_Robot_Count>=9) AND
							MAIN.R9.EL6695_PortC_MissingLink;
		Out_To_ICxx.System_Faults[819]:=Fault_Tmrs[819].Q;
	(*Fault820 - R10 EK1100 Out Port Cabe disconnected*)
		Fault_Tmrs[820].PT:=No_Timer;
		Fault_Tmrs[820]();
		Fault_Tmrs[820].IN:= (GTAC_CONFIG.Option_Robot_Count>=10) AND
							MAIN.R10.EL6695_PortC_MissingLink;
		Out_To_ICxx.System_Faults[820]:=Fault_Tmrs[820].Q;
	(*Fault821 - R11 EK1100 Out Port Cabe disconnected*)
		Fault_Tmrs[821].PT:=No_Timer;
		Fault_Tmrs[821]();
		Fault_Tmrs[821].IN:= (GTAC_CONFIG.Option_Robot_Count>=11) AND
							MAIN.R11.EL6695_PortC_MissingLink;
		Out_To_ICxx.System_Faults[821]:=Fault_Tmrs[821].Q;
	(*Fault822 - R12 EK1100 Out Port Cabe disconnected*)
		Fault_Tmrs[822].PT:=No_Timer;
		Fault_Tmrs[822]();
		Fault_Tmrs[822].IN:= (GTAC_CONFIG.Option_Robot_Count>=12) AND
							MAIN.R12.EL6695_PortC_MissingLink;
		Out_To_ICxx.System_Faults[822]:=Fault_Tmrs[822].Q;
	(*Fault823 - R13 EK1100 Out Port Cabe disconnected*)
		Fault_Tmrs[823].PT:=No_Timer;
		Fault_Tmrs[823]();
		Fault_Tmrs[823].IN:= (GTAC_CONFIG.Option_Robot_Count>=13) AND
							MAIN.R13.EL6695_PortC_MissingLink;
		Out_To_ICxx.System_Faults[823]:=Fault_Tmrs[823].Q;
	(*Fault824 - R14 EK1100 Out Port Cabe disconnected*)
		Fault_Tmrs[824].PT:=No_Timer;
		Fault_Tmrs[824]();
		Fault_Tmrs[824].IN:= (GTAC_CONFIG.Option_Robot_Count>=14) AND
							MAIN.R14.EL6695_PortC_MissingLink;
		Out_To_ICxx.System_Faults[824]:=Fault_Tmrs[824].Q;
	(*Fault825 - R15 EK1100 Out Port Cabe disconnected*)
		Fault_Tmrs[825].PT:=No_Timer;
		Fault_Tmrs[825]();
		Fault_Tmrs[825].IN:= (GTAC_CONFIG.Option_Robot_Count>=15) AND
							MAIN.R15.EL6695_PortC_MissingLink;
		Out_To_ICxx.System_Faults[825]:=Fault_Tmrs[825].Q;
	(*Fault826 - R16 EK1100 Out Port Cabe disconnected*)
		Fault_Tmrs[826].PT:=No_Timer;
		Fault_Tmrs[826]();
		Fault_Tmrs[826].IN:= (GTAC_CONFIG.Option_Robot_Count>=16) AND
							MAIN.R16.EL6695_PortC_MissingLink;
		Out_To_ICxx.System_Faults[826]:=Fault_Tmrs[826].Q;
	(*Fault827 - R17 EK1100 Out Port Cabe disconnected*)
		Fault_Tmrs[827].PT:=No_Timer;
		Fault_Tmrs[827]();
		Fault_Tmrs[827].IN:= (GTAC_CONFIG.Option_Robot_Count>=17) AND
							MAIN.R17.EL6695_PortC_MissingLink;
		Out_To_ICxx.System_Faults[827]:=Fault_Tmrs[827].Q;
	(*Fault828 - R18 EK1100 Out Port Cabe disconnected*)
		Fault_Tmrs[828].PT:=No_Timer;
		Fault_Tmrs[828]();
		Fault_Tmrs[828].IN:= (GTAC_CONFIG.Option_Robot_Count>=18) AND
							MAIN.R18.EL6695_PortC_MissingLink;
		Out_To_ICxx.System_Faults[828]:=Fault_Tmrs[828].Q;
	(*Fault829 - R19 EK1100 Out Port Cabe disconnected*)
		Fault_Tmrs[829].PT:=No_Timer;
		Fault_Tmrs[829]();
		Fault_Tmrs[829].IN:= (GTAC_CONFIG.Option_Robot_Count>=19) AND
							MAIN.R19.EL6695_PortC_MissingLink;
		Out_To_ICxx.System_Faults[829]:=Fault_Tmrs[829].Q;
	(*Fault830 - R20 EK1100 Out Port Cabe disconnected*)
		Fault_Tmrs[830].PT:=No_Timer;
		Fault_Tmrs[830]();
		Fault_Tmrs[830].IN:= (GTAC_CONFIG.Option_Robot_Count>=20) AND
							MAIN.R20.EL6695_PortC_MissingLink;
		Out_To_ICxx.System_Faults[830]:=Fault_Tmrs[830].Q;
	(*Fault831 - R21 EK1100 Out Port Cabe disconnected*)
		Fault_Tmrs[831].PT:=No_Timer;
		Fault_Tmrs[831]();
		Fault_Tmrs[831].IN:= (GTAC_CONFIG.Option_Robot_Count>=21) AND
							MAIN.R21.EL6695_PortC_MissingLink;
		Out_To_ICxx.System_Faults[831]:=Fault_Tmrs[831].Q;
	(*Fault832 - R22 EK1100 Out Port Cabe disconnected*)
		Fault_Tmrs[832].PT:=No_Timer;
		Fault_Tmrs[832]();
		Fault_Tmrs[832].IN:= (GTAC_CONFIG.Option_Robot_Count>=22) AND
							MAIN.R22.EL6695_PortC_MissingLink;
		Out_To_ICxx.System_Faults[832]:=Fault_Tmrs[832].Q;
	(*Fault833 - R23 EK1100 Out Port Cabe disconnected*)
		Fault_Tmrs[833].PT:=No_Timer;
		Fault_Tmrs[833]();
		Fault_Tmrs[833].IN:= (GTAC_CONFIG.Option_Robot_Count>=23) AND
							MAIN.R23.EL6695_PortC_MissingLink;
		Out_To_ICxx.System_Faults[833]:=Fault_Tmrs[833].Q;
	(*Fault834 - R24 EK1100 Out Port Cabe disconnected*)
		Fault_Tmrs[834].PT:=No_Timer;
		Fault_Tmrs[834]();
		Fault_Tmrs[834].IN:= (GTAC_CONFIG.Option_Robot_Count>=24) AND
							MAIN.R24.EL6695_PortC_MissingLink;
		Out_To_ICxx.System_Faults[834]:=Fault_Tmrs[834].Q;
	(*Fault835 - R25 EK1100 Out Port Cabe disconnected*)
		Fault_Tmrs[835].PT:=No_Timer;
		Fault_Tmrs[835]();
		Fault_Tmrs[835].IN:= (GTAC_CONFIG.Option_Robot_Count>=25) AND
							MAIN.R25.EL6695_PortC_MissingLink;
		Out_To_ICxx.System_Faults[835]:=Fault_Tmrs[835].Q;
	(*Fault836 - R26 EK1100 Out Port Cabe disconnected*)
		Fault_Tmrs[836].PT:=No_Timer;
		Fault_Tmrs[836]();
		Fault_Tmrs[836].IN:= (GTAC_CONFIG.Option_Robot_Count>=26) AND
							MAIN.R26.EL6695_PortC_MissingLink;
		Out_To_ICxx.System_Faults[836]:=Fault_Tmrs[836].Q;
	(*Fault837 - R27 EK1100 Out Port Cabe disconnected*)
		Fault_Tmrs[837].PT:=No_Timer;
		Fault_Tmrs[837]();
		Fault_Tmrs[837].IN:= (GTAC_CONFIG.Option_Robot_Count>=27) AND
							MAIN.R27.EL6695_PortC_MissingLink;
		Out_To_ICxx.System_Faults[837]:=Fault_Tmrs[837].Q;
	(*Fault838 - R28 EK1100 Out Port Cabe disconnected*)
		Fault_Tmrs[838].PT:=No_Timer;
		Fault_Tmrs[838]();
		Fault_Tmrs[838].IN:= (GTAC_CONFIG.Option_Robot_Count>=28) AND
							MAIN.R28.EL6695_PortC_MissingLink;
		Out_To_ICxx.System_Faults[838]:=Fault_Tmrs[838].Q;
	(*Fault839 - R29 EK1100 Out Port Cabe disconnected*)
		Fault_Tmrs[839].PT:=No_Timer;
		Fault_Tmrs[839]();
		Fault_Tmrs[839].IN:= (GTAC_CONFIG.Option_Robot_Count>=29) AND
							MAIN.R29.EL6695_PortC_MissingLink;
		Out_To_ICxx.System_Faults[839]:=Fault_Tmrs[839].Q;
	(*Fault840 - R30 EK1100 Out Port Cabe disconnected*)
		Fault_Tmrs[840].PT:=No_Timer;
		Fault_Tmrs[840]();
		Fault_Tmrs[840].IN:= (GTAC_CONFIG.Option_Robot_Count>=30) AND
							MAIN.R30.EL6695_PortC_MissingLink;
		Out_To_ICxx.System_Faults[840]:=Fault_Tmrs[840].Q;

	(*-----Internal Cable(s)-------*)
	(*Fault841 - R01 Internal Cable(s) disconnected*)
		Fault_Tmrs[841].PT:=No_Timer;
		Fault_Tmrs[841]();
		Fault_Tmrs[841].IN:= (GTAC_CONFIG.Option_Robot_Count>=1) AND
							MAIN.R1.EK1100_PortC_MissingLink;
		Out_To_ICxx.System_Faults[841]:=Fault_Tmrs[841].Q;
	(*Fault842 - R02 Internal Cable(s) disconnected*)
		Fault_Tmrs[842].PT:=No_Timer;
		Fault_Tmrs[842]();
		Fault_Tmrs[842].IN:= (GTAC_CONFIG.Option_Robot_Count>=2) AND
							MAIN.R2.EK1100_PortC_MissingLink;
		Out_To_ICxx.System_Faults[842]:=Fault_Tmrs[842].Q;
	(*Fault843 - R03 Internal Cable(s) disconnected*)
		Fault_Tmrs[843].PT:=No_Timer;
		Fault_Tmrs[843]();
		Fault_Tmrs[843].IN:= (GTAC_CONFIG.Option_Robot_Count>=3) AND
							MAIN.R3.EK1100_PortC_MissingLink;
		Out_To_ICxx.System_Faults[843]:=Fault_Tmrs[843].Q;
	(*Fault844 - R04 Internal Cable(s) disconnected*)
		Fault_Tmrs[844].PT:=No_Timer;
		Fault_Tmrs[844]();
		Fault_Tmrs[844].IN:= (GTAC_CONFIG.Option_Robot_Count>=4) AND
							MAIN.R4.EK1100_PortC_MissingLink;
		Out_To_ICxx.System_Faults[844]:=Fault_Tmrs[844].Q;
	(*Fault845 - R05 Internal Cable(s) disconnected*)
		Fault_Tmrs[845].PT:=No_Timer;
		Fault_Tmrs[845]();
		Fault_Tmrs[845].IN:= (GTAC_CONFIG.Option_Robot_Count>=5) AND
							MAIN.R5.EK1100_PortC_MissingLink;
		Out_To_ICxx.System_Faults[845]:=Fault_Tmrs[845].Q;
	(*Fault846 - R06 Internal Cable(s) disconnected*)
		Fault_Tmrs[846].PT:=No_Timer;
		Fault_Tmrs[846]();
		Fault_Tmrs[846].IN:= (GTAC_CONFIG.Option_Robot_Count>=6) AND
							MAIN.R6.EK1100_PortC_MissingLink;
		Out_To_ICxx.System_Faults[846]:=Fault_Tmrs[846].Q;
	(*Fault847 - R07 Internal Cable(s) disconnected*)
		Fault_Tmrs[847].PT:=No_Timer;
		Fault_Tmrs[847]();
		Fault_Tmrs[847].IN:= (GTAC_CONFIG.Option_Robot_Count>=7) AND
							MAIN.R7.EK1100_PortC_MissingLink;
		Out_To_ICxx.System_Faults[847]:=Fault_Tmrs[847].Q;
	(*Fault848 - R08 Internal Cable(s) disconnected*)
		Fault_Tmrs[848].PT:=No_Timer;
		Fault_Tmrs[848]();
		Fault_Tmrs[848].IN:= (GTAC_CONFIG.Option_Robot_Count>=8) AND
							MAIN.R8.EK1100_PortC_MissingLink;
		Out_To_ICxx.System_Faults[848]:=Fault_Tmrs[848].Q;
	(*Fault849 - R09 Internal Cable(s) disconnected*)
		Fault_Tmrs[849].PT:=No_Timer;
		Fault_Tmrs[849]();
		Fault_Tmrs[849].IN:= (GTAC_CONFIG.Option_Robot_Count>=9) AND
							MAIN.R9.EK1100_PortC_MissingLink;
		Out_To_ICxx.System_Faults[849]:=Fault_Tmrs[849].Q;
	(*Fault850 - R10 Internal Cable(s) disconnected*)
		Fault_Tmrs[850].PT:=No_Timer;
		Fault_Tmrs[850]();
		Fault_Tmrs[850].IN:= (GTAC_CONFIG.Option_Robot_Count>=10) AND
							MAIN.R10.EK1100_PortC_MissingLink;
		Out_To_ICxx.System_Faults[850]:=Fault_Tmrs[850].Q;
	(*Fault851 - R11 Internal Cable(s) disconnected*)
		Fault_Tmrs[851].PT:=No_Timer;
		Fault_Tmrs[851]();
		Fault_Tmrs[851].IN:= (GTAC_CONFIG.Option_Robot_Count>=11) AND
							MAIN.R11.EK1100_PortC_MissingLink;
		Out_To_ICxx.System_Faults[851]:=Fault_Tmrs[851].Q;
	(*Fault852 - R12 Internal Cable(s) disconnected*)
		Fault_Tmrs[852].PT:=No_Timer;
		Fault_Tmrs[852]();
		Fault_Tmrs[852].IN:= (GTAC_CONFIG.Option_Robot_Count>=12) AND
							MAIN.R12.EK1100_PortC_MissingLink;
		Out_To_ICxx.System_Faults[852]:=Fault_Tmrs[852].Q;
	(*Fault853 - R13 Internal Cable(s) disconnected*)
		Fault_Tmrs[853].PT:=No_Timer;
		Fault_Tmrs[853]();
		Fault_Tmrs[853].IN:= (GTAC_CONFIG.Option_Robot_Count>=13) AND
							MAIN.R13.EK1100_PortC_MissingLink;
		Out_To_ICxx.System_Faults[853]:=Fault_Tmrs[853].Q;
	(*Fault854 - R14 Internal Cable(s) disconnected*)
		Fault_Tmrs[854].PT:=No_Timer;
		Fault_Tmrs[854]();
		Fault_Tmrs[854].IN:= (GTAC_CONFIG.Option_Robot_Count>=14) AND
							MAIN.R14.EK1100_PortC_MissingLink;
		Out_To_ICxx.System_Faults[854]:=Fault_Tmrs[854].Q;
	(*Fault855 - R15 Internal Cable(s) disconnected*)
		Fault_Tmrs[855].PT:=No_Timer;
		Fault_Tmrs[855]();
		Fault_Tmrs[855].IN:= (GTAC_CONFIG.Option_Robot_Count>=15) AND
							MAIN.R15.EK1100_PortC_MissingLink;
		Out_To_ICxx.System_Faults[855]:=Fault_Tmrs[855].Q;
	(*Fault856 - R16 Internal Cable(s) disconnected*)
		Fault_Tmrs[856].PT:=No_Timer;
		Fault_Tmrs[856]();
		Fault_Tmrs[856].IN:= (GTAC_CONFIG.Option_Robot_Count>=16) AND
							MAIN.R16.EK1100_PortC_MissingLink;
		Out_To_ICxx.System_Faults[856]:=Fault_Tmrs[856].Q;
	(*Fault857 - R17 Internal Cable(s) disconnected*)
		Fault_Tmrs[857].PT:=No_Timer;
		Fault_Tmrs[857]();
		Fault_Tmrs[857].IN:= (GTAC_CONFIG.Option_Robot_Count>=17) AND
							MAIN.R17.EK1100_PortC_MissingLink;
		Out_To_ICxx.System_Faults[857]:=Fault_Tmrs[857].Q;
	(*Fault858 - R18 Internal Cable(s) disconnected*)
		Fault_Tmrs[858].PT:=No_Timer;
		Fault_Tmrs[858]();
		Fault_Tmrs[858].IN:= (GTAC_CONFIG.Option_Robot_Count>=18) AND
							MAIN.R18.EK1100_PortC_MissingLink;
		Out_To_ICxx.System_Faults[858]:=Fault_Tmrs[858].Q;
	(*Fault859 - R19 Internal Cable(s) disconnected*)
		Fault_Tmrs[859].PT:=No_Timer;
		Fault_Tmrs[859]();
		Fault_Tmrs[859].IN:= (GTAC_CONFIG.Option_Robot_Count>=19) AND
							MAIN.R19.EK1100_PortC_MissingLink;
		Out_To_ICxx.System_Faults[859]:=Fault_Tmrs[859].Q;
	(*Fault860 - R20 Internal Cable(s) disconnected*)
		Fault_Tmrs[860].PT:=No_Timer;
		Fault_Tmrs[860]();
		Fault_Tmrs[860].IN:= (GTAC_CONFIG.Option_Robot_Count>=20) AND
							MAIN.R20.EK1100_PortC_MissingLink;
		Out_To_ICxx.System_Faults[860]:=Fault_Tmrs[860].Q;
	(*Fault861 - R21 Internal Cable(s) disconnected*)
		Fault_Tmrs[861].PT:=No_Timer;
		Fault_Tmrs[861]();
		Fault_Tmrs[861].IN:= (GTAC_CONFIG.Option_Robot_Count>=21) AND
							MAIN.R21.EK1100_PortC_MissingLink;
		Out_To_ICxx.System_Faults[861]:=Fault_Tmrs[861].Q;
	(*Fault862 - R22 Internal Cable(s) disconnected*)
		Fault_Tmrs[862].PT:=No_Timer;
		Fault_Tmrs[862]();
		Fault_Tmrs[862].IN:= (GTAC_CONFIG.Option_Robot_Count>=22) AND
							MAIN.R22.EK1100_PortC_MissingLink;
		Out_To_ICxx.System_Faults[862]:=Fault_Tmrs[862].Q;
	(*Fault863 - R23 Internal Cable(s) disconnected*)
		Fault_Tmrs[863].PT:=No_Timer;
		Fault_Tmrs[863]();
		Fault_Tmrs[863].IN:= (GTAC_CONFIG.Option_Robot_Count>=23) AND
							MAIN.R23.EK1100_PortC_MissingLink;
		Out_To_ICxx.System_Faults[863]:=Fault_Tmrs[863].Q;
	(*Fault864 - R24 Internal Cable(s) disconnected*)
		Fault_Tmrs[864].PT:=No_Timer;
		Fault_Tmrs[864]();
		Fault_Tmrs[864].IN:= (GTAC_CONFIG.Option_Robot_Count>=24) AND
							MAIN.R24.EK1100_PortC_MissingLink;
		Out_To_ICxx.System_Faults[864]:=Fault_Tmrs[864].Q;
	(*Fault865 - R25 Internal Cable(s) disconnected*)
		Fault_Tmrs[865].PT:=No_Timer;
		Fault_Tmrs[865]();
		Fault_Tmrs[865].IN:= (GTAC_CONFIG.Option_Robot_Count>=25) AND
							MAIN.R25.EK1100_PortC_MissingLink;
		Out_To_ICxx.System_Faults[865]:=Fault_Tmrs[865].Q;
	(*Fault866 - R26 Internal Cable(s) disconnected*)
		Fault_Tmrs[866].PT:=No_Timer;
		Fault_Tmrs[866]();
		Fault_Tmrs[866].IN:= (GTAC_CONFIG.Option_Robot_Count>=26) AND
							MAIN.R26.EK1100_PortC_MissingLink;
		Out_To_ICxx.System_Faults[866]:=Fault_Tmrs[866].Q;
	(*Fault867 - R27 Internal Cable(s) disconnected*)
		Fault_Tmrs[867].PT:=No_Timer;
		Fault_Tmrs[867]();
		Fault_Tmrs[867].IN:= (GTAC_CONFIG.Option_Robot_Count>=27) AND
							MAIN.R27.EK1100_PortC_MissingLink;
		Out_To_ICxx.System_Faults[867]:=Fault_Tmrs[867].Q;
	(*Fault868 - R28 Internal Cable(s) disconnected*)
		Fault_Tmrs[868].PT:=No_Timer;
		Fault_Tmrs[868]();
		Fault_Tmrs[868].IN:= (GTAC_CONFIG.Option_Robot_Count>=28) AND
							MAIN.R28.EK1100_PortC_MissingLink;
		Out_To_ICxx.System_Faults[868]:=Fault_Tmrs[868].Q;
	(*Fault869 - R29 Internal Cable(s) disconnected*)
		Fault_Tmrs[869].PT:=No_Timer;
		Fault_Tmrs[869]();
		Fault_Tmrs[869].IN:= (GTAC_CONFIG.Option_Robot_Count>=29) AND
							MAIN.R29.EK1100_PortC_MissingLink;
		Out_To_ICxx.System_Faults[869]:=Fault_Tmrs[869].Q;
	(*Fault870 - R30 Internal Cable(s) disconnected*)
		Fault_Tmrs[870].PT:=No_Timer;
		Fault_Tmrs[870]();
		Fault_Tmrs[870].IN:= (GTAC_CONFIG.Option_Robot_Count>=30) AND
							MAIN.R30.EK1100_PortC_MissingLink;
		Out_To_ICxx.System_Faults[870]:=Fault_Tmrs[870].Q;

	(*-----Water Stand Cable(s)-------*)
	(*Fault871 - R01 Water Stand Cable(s) disconnected*)
		Fault_Tmrs[871].PT:=No_Timer;
		Fault_Tmrs[871]();
		Fault_Tmrs[871].IN:= (GTAC_CONFIG.Option_Robot_Count>=1) AND
							(MAIN.R1.EK1122_PortD_MissingLink
							OR (MAIN.R1.WS[1].ECatSlave_Cable_Breaks<>0) OR (MAIN.R1.WS[2].ECatSlave_Cable_Breaks<>0));
		Out_To_ICxx.System_Faults[871]:=Fault_Tmrs[871].Q;
	(*Fault872 - R02 Water Stand Cable(s) disconnected*)
		Fault_Tmrs[872].PT:=No_Timer;
		Fault_Tmrs[872]();
		Fault_Tmrs[872].IN:= (GTAC_CONFIG.Option_Robot_Count>=2) AND
							(MAIN.R2.EK1122_PortD_MissingLink
							OR (MAIN.R2.WS[1].ECatSlave_Cable_Breaks<>0) OR (MAIN.R2.WS[2].ECatSlave_Cable_Breaks<>0));
		Out_To_ICxx.System_Faults[872]:=Fault_Tmrs[872].Q;
	(*Fault873 - R03 Water Stand Cable(s) disconnected*)
		Fault_Tmrs[873].PT:=No_Timer;
		Fault_Tmrs[873]();
		Fault_Tmrs[873].IN:= (GTAC_CONFIG.Option_Robot_Count>=3) AND
							(MAIN.R3.EK1122_PortD_MissingLink
							OR (MAIN.R3.WS[1].ECatSlave_Cable_Breaks<>0) OR (MAIN.R3.WS[2].ECatSlave_Cable_Breaks<>0));
		Out_To_ICxx.System_Faults[873]:=Fault_Tmrs[873].Q;
	(*Fault874 - R04 Water Stand Cable(s) disconnected*)
		Fault_Tmrs[874].PT:=No_Timer;
		Fault_Tmrs[874]();
		Fault_Tmrs[874].IN:= (GTAC_CONFIG.Option_Robot_Count>=4) AND
							(MAIN.R4.EK1122_PortD_MissingLink
							OR (MAIN.R4.WS[1].ECatSlave_Cable_Breaks<>0) OR (MAIN.R4.WS[2].ECatSlave_Cable_Breaks<>0));
		Out_To_ICxx.System_Faults[874]:=Fault_Tmrs[874].Q;
	(*Fault875 - R05 Water Stand Cable(s) disconnected*)
		Fault_Tmrs[875].PT:=No_Timer;
		Fault_Tmrs[875]();
		Fault_Tmrs[875].IN:= (GTAC_CONFIG.Option_Robot_Count>=5) AND
							(MAIN.R5.EK1122_PortD_MissingLink
							OR (MAIN.R5.WS[1].ECatSlave_Cable_Breaks<>0) OR (MAIN.R5.WS[2].ECatSlave_Cable_Breaks<>0));
		Out_To_ICxx.System_Faults[875]:=Fault_Tmrs[875].Q;
	(*Fault876 - R06 Water Stand Cable(s) disconnected*)
		Fault_Tmrs[876].PT:=No_Timer;
		Fault_Tmrs[876]();
		Fault_Tmrs[876].IN:= (GTAC_CONFIG.Option_Robot_Count>=6) AND
							(MAIN.R6.EK1122_PortD_MissingLink
							OR (MAIN.R6.WS[1].ECatSlave_Cable_Breaks<>0) OR (MAIN.R6.WS[2].ECatSlave_Cable_Breaks<>0));
		Out_To_ICxx.System_Faults[876]:=Fault_Tmrs[876].Q;
	(*Fault877 - R07 Water Stand Cable(s) disconnected*)
		Fault_Tmrs[877].PT:=No_Timer;
		Fault_Tmrs[877]();
		Fault_Tmrs[877].IN:= (GTAC_CONFIG.Option_Robot_Count>=7) AND
							(MAIN.R7.EK1122_PortD_MissingLink
							OR (MAIN.R7.WS[1].ECatSlave_Cable_Breaks<>0) OR (MAIN.R7.WS[2].ECatSlave_Cable_Breaks<>0));
		Out_To_ICxx.System_Faults[877]:=Fault_Tmrs[877].Q;
	(*Fault878 - R08 Water Stand Cable(s) disconnected*)
		Fault_Tmrs[878].PT:=No_Timer;
		Fault_Tmrs[878]();
		Fault_Tmrs[878].IN:= (GTAC_CONFIG.Option_Robot_Count>=8) AND
							(MAIN.R8.EK1122_PortD_MissingLink
							OR (MAIN.R8.WS[1].ECatSlave_Cable_Breaks<>0) OR (MAIN.R8.WS[2].ECatSlave_Cable_Breaks<>0));
		Out_To_ICxx.System_Faults[878]:=Fault_Tmrs[878].Q;
	(*Fault879 - R09 Water Stand Cable(s) disconnected*)
		Fault_Tmrs[879].PT:=No_Timer;
		Fault_Tmrs[879]();
		Fault_Tmrs[879].IN:= (GTAC_CONFIG.Option_Robot_Count>=9) AND
							(MAIN.R9.EK1122_PortD_MissingLink
							OR (MAIN.R9.WS[1].ECatSlave_Cable_Breaks<>0) OR (MAIN.R9.WS[2].ECatSlave_Cable_Breaks<>0));
		Out_To_ICxx.System_Faults[879]:=Fault_Tmrs[879].Q;
	(*Fault880 - R10 Water Stand Cable(s) disconnected*)
		Fault_Tmrs[880].PT:=No_Timer;
		Fault_Tmrs[880]();
		Fault_Tmrs[880].IN:= (GTAC_CONFIG.Option_Robot_Count>=10) AND
							(MAIN.R10.EK1122_PortD_MissingLink
							OR (MAIN.R10.WS[1].ECatSlave_Cable_Breaks<>0) OR (MAIN.R10.WS[2].ECatSlave_Cable_Breaks<>0));
		Out_To_ICxx.System_Faults[880]:=Fault_Tmrs[880].Q;
	(*Fault881 - R11 Water Stand Cable(s) disconnected*)
		Fault_Tmrs[881].PT:=No_Timer;
		Fault_Tmrs[881]();
		Fault_Tmrs[881].IN:= (GTAC_CONFIG.Option_Robot_Count>=11) AND
							(MAIN.R11.EK1122_PortD_MissingLink
							OR (MAIN.R11.WS[1].ECatSlave_Cable_Breaks<>0) OR (MAIN.R11.WS[2].ECatSlave_Cable_Breaks<>0));
		Out_To_ICxx.System_Faults[881]:=Fault_Tmrs[881].Q;
	(*Fault882 - R12 Water Stand Cable(s) disconnected*)
		Fault_Tmrs[882].PT:=No_Timer;
		Fault_Tmrs[882]();
		Fault_Tmrs[882].IN:= (GTAC_CONFIG.Option_Robot_Count>=12) AND
							(MAIN.R12.EK1122_PortD_MissingLink
							OR (MAIN.R12.WS[1].ECatSlave_Cable_Breaks<>0) OR (MAIN.R12.WS[2].ECatSlave_Cable_Breaks<>0));
		Out_To_ICxx.System_Faults[882]:=Fault_Tmrs[882].Q;
	(*Fault883 - R13 Water Stand Cable(s) disconnected*)
		Fault_Tmrs[883].PT:=No_Timer;
		Fault_Tmrs[883]();
		Fault_Tmrs[883].IN:= (GTAC_CONFIG.Option_Robot_Count>=13) AND
							(MAIN.R13.EK1122_PortD_MissingLink
							OR (MAIN.R13.WS[1].ECatSlave_Cable_Breaks<>0) OR (MAIN.R13.WS[2].ECatSlave_Cable_Breaks<>0));
		Out_To_ICxx.System_Faults[883]:=Fault_Tmrs[883].Q;
	(*Fault884 - R14 Water Stand Cable(s) disconnected*)
		Fault_Tmrs[884].PT:=No_Timer;
		Fault_Tmrs[884]();
		Fault_Tmrs[884].IN:= (GTAC_CONFIG.Option_Robot_Count>=14) AND
							(MAIN.R14.EK1122_PortD_MissingLink
							OR (MAIN.R14.WS[1].ECatSlave_Cable_Breaks<>0) OR (MAIN.R14.WS[2].ECatSlave_Cable_Breaks<>0));
		Out_To_ICxx.System_Faults[884]:=Fault_Tmrs[884].Q;
	(*Fault885 - R15 Water Stand Cable(s) disconnected*)
		Fault_Tmrs[885].PT:=No_Timer;
		Fault_Tmrs[885]();
		Fault_Tmrs[885].IN:= (GTAC_CONFIG.Option_Robot_Count>=15) AND
							(MAIN.R15.EK1122_PortD_MissingLink
							OR (MAIN.R15.WS[1].ECatSlave_Cable_Breaks<>0) OR (MAIN.R15.WS[2].ECatSlave_Cable_Breaks<>0));
		Out_To_ICxx.System_Faults[885]:=Fault_Tmrs[885].Q;
	(*Fault886 - R16 Water Stand Cable(s) disconnected*)
		Fault_Tmrs[886].PT:=No_Timer;
		Fault_Tmrs[886]();
		Fault_Tmrs[886].IN:= (GTAC_CONFIG.Option_Robot_Count>=16) AND
							(MAIN.R16.EK1122_PortD_MissingLink
							OR (MAIN.R16.WS[1].ECatSlave_Cable_Breaks<>0) OR (MAIN.R16.WS[2].ECatSlave_Cable_Breaks<>0));
		Out_To_ICxx.System_Faults[886]:=Fault_Tmrs[886].Q;
	(*Fault887 - R17 Water Stand Cable(s) disconnected*)
		Fault_Tmrs[887].PT:=No_Timer;
		Fault_Tmrs[887]();
		Fault_Tmrs[887].IN:= (GTAC_CONFIG.Option_Robot_Count>=17) AND
							(MAIN.R17.EK1122_PortD_MissingLink
							OR (MAIN.R17.WS[1].ECatSlave_Cable_Breaks<>0) OR (MAIN.R17.WS[2].ECatSlave_Cable_Breaks<>0));
		Out_To_ICxx.System_Faults[887]:=Fault_Tmrs[887].Q;
	(*Fault888 - R18 Water Stand Cable(s) disconnected*)
		Fault_Tmrs[888].PT:=No_Timer;
		Fault_Tmrs[888]();
		Fault_Tmrs[888].IN:= (GTAC_CONFIG.Option_Robot_Count>=18) AND
							(MAIN.R18.EK1122_PortD_MissingLink
							OR (MAIN.R18.WS[1].ECatSlave_Cable_Breaks<>0) OR (MAIN.R18.WS[2].ECatSlave_Cable_Breaks<>0));
		Out_To_ICxx.System_Faults[888]:=Fault_Tmrs[888].Q;
	(*Fault889 - R19 Water Stand Cable(s) disconnected*)
		Fault_Tmrs[889].PT:=No_Timer;
		Fault_Tmrs[889]();
		Fault_Tmrs[889].IN:= (GTAC_CONFIG.Option_Robot_Count>=19) AND
							(MAIN.R19.EK1122_PortD_MissingLink
							OR (MAIN.R19.WS[1].ECatSlave_Cable_Breaks<>0) OR (MAIN.R19.WS[2].ECatSlave_Cable_Breaks<>0));
		Out_To_ICxx.System_Faults[889]:=Fault_Tmrs[889].Q;
	(*Fault890 - R20 Water Stand Cable(s) disconnected*)
		Fault_Tmrs[890].PT:=No_Timer;
		Fault_Tmrs[890]();
		Fault_Tmrs[890].IN:= (GTAC_CONFIG.Option_Robot_Count>=20) AND
							(MAIN.R20.EK1122_PortD_MissingLink
							OR (MAIN.R20.WS[1].ECatSlave_Cable_Breaks<>0) OR (MAIN.R20.WS[2].ECatSlave_Cable_Breaks<>0));
		Out_To_ICxx.System_Faults[890]:=Fault_Tmrs[890].Q;
	(*Fault891 - R21 Water Stand Cable(s) disconnected*)
		Fault_Tmrs[891].PT:=No_Timer;
		Fault_Tmrs[891]();
		Fault_Tmrs[891].IN:= (GTAC_CONFIG.Option_Robot_Count>=21) AND
							(MAIN.R21.EK1122_PortD_MissingLink
							OR (MAIN.R21.WS[1].ECatSlave_Cable_Breaks<>0) OR (MAIN.R21.WS[2].ECatSlave_Cable_Breaks<>0));
		Out_To_ICxx.System_Faults[891]:=Fault_Tmrs[891].Q;
	(*Fault892 - R22 Water Stand Cable(s) disconnected*)
		Fault_Tmrs[892].PT:=No_Timer;
		Fault_Tmrs[892]();
		Fault_Tmrs[892].IN:= (GTAC_CONFIG.Option_Robot_Count>=22) AND
							(MAIN.R22.EK1122_PortD_MissingLink
							OR (MAIN.R22.WS[1].ECatSlave_Cable_Breaks<>0) OR (MAIN.R22.WS[2].ECatSlave_Cable_Breaks<>0));
		Out_To_ICxx.System_Faults[892]:=Fault_Tmrs[892].Q;
	(*Fault893 - R23 Water Stand Cable(s) disconnected*)
		Fault_Tmrs[893].PT:=No_Timer;
		Fault_Tmrs[893]();
		Fault_Tmrs[893].IN:= (GTAC_CONFIG.Option_Robot_Count>=23) AND
							(MAIN.R23.EK1122_PortD_MissingLink
							OR (MAIN.R23.WS[1].ECatSlave_Cable_Breaks<>0) OR (MAIN.R23.WS[2].ECatSlave_Cable_Breaks<>0));
		Out_To_ICxx.System_Faults[893]:=Fault_Tmrs[893].Q;
	(*Fault894 - R24 Water Stand Cable(s) disconnected*)
		Fault_Tmrs[894].PT:=No_Timer;
		Fault_Tmrs[894]();
		Fault_Tmrs[894].IN:= (GTAC_CONFIG.Option_Robot_Count>=24) AND
							(MAIN.R24.EK1122_PortD_MissingLink
							OR (MAIN.R24.WS[1].ECatSlave_Cable_Breaks<>0) OR (MAIN.R24.WS[2].ECatSlave_Cable_Breaks<>0));
		Out_To_ICxx.System_Faults[894]:=Fault_Tmrs[894].Q;
	(*Fault895 - R25 Water Stand Cable(s) disconnected*)
		Fault_Tmrs[895].PT:=No_Timer;
		Fault_Tmrs[895]();
		Fault_Tmrs[895].IN:= (GTAC_CONFIG.Option_Robot_Count>=25) AND
							(MAIN.R25.EK1122_PortD_MissingLink
							OR (MAIN.R25.WS[1].ECatSlave_Cable_Breaks<>0) OR (MAIN.R25.WS[2].ECatSlave_Cable_Breaks<>0));
		Out_To_ICxx.System_Faults[895]:=Fault_Tmrs[895].Q;
	(*Fault896 - R26 Water Stand Cable(s) disconnected*)
		Fault_Tmrs[896].PT:=No_Timer;
		Fault_Tmrs[896]();
		Fault_Tmrs[896].IN:= (GTAC_CONFIG.Option_Robot_Count>=26) AND
							(MAIN.R26.EK1122_PortD_MissingLink
							OR (MAIN.R26.WS[1].ECatSlave_Cable_Breaks<>0) OR (MAIN.R26.WS[2].ECatSlave_Cable_Breaks<>0));
		Out_To_ICxx.System_Faults[896]:=Fault_Tmrs[896].Q;
	(*Fault897 - R27 Water Stand Cable(s) disconnected*)
		Fault_Tmrs[897].PT:=No_Timer;
		Fault_Tmrs[897]();
		Fault_Tmrs[897].IN:= (GTAC_CONFIG.Option_Robot_Count>=27) AND
							(MAIN.R27.EK1122_PortD_MissingLink
							OR (MAIN.R27.WS[1].ECatSlave_Cable_Breaks<>0) OR (MAIN.R27.WS[2].ECatSlave_Cable_Breaks<>0));
		Out_To_ICxx.System_Faults[897]:=Fault_Tmrs[897].Q;
	(*Fault898 - R28 Water Stand Cable(s) disconnected*)
		Fault_Tmrs[898].PT:=No_Timer;
		Fault_Tmrs[898]();
		Fault_Tmrs[898].IN:= (GTAC_CONFIG.Option_Robot_Count>=28) AND
							(MAIN.R28.EK1122_PortD_MissingLink
							OR (MAIN.R28.WS[1].ECatSlave_Cable_Breaks<>0) OR (MAIN.R28.WS[2].ECatSlave_Cable_Breaks<>0));
		Out_To_ICxx.System_Faults[898]:=Fault_Tmrs[898].Q;
	(*Fault899 - R29 Water Stand Cable(s) disconnected*)
		Fault_Tmrs[899].PT:=No_Timer;
		Fault_Tmrs[899]();
		Fault_Tmrs[899].IN:= (GTAC_CONFIG.Option_Robot_Count>=29) AND
							(MAIN.R29.EK1122_PortD_MissingLink
							OR (MAIN.R29.WS[1].ECatSlave_Cable_Breaks<>0) OR (MAIN.R29.WS[2].ECatSlave_Cable_Breaks<>0));
		Out_To_ICxx.System_Faults[899]:=Fault_Tmrs[899].Q;
	(*Fault900 - R30 Water Stand Cable(s) disconnected*)
		Fault_Tmrs[900].PT:=No_Timer;
		Fault_Tmrs[900]();
		Fault_Tmrs[900].IN:= (GTAC_CONFIG.Option_Robot_Count>=30) AND
							(MAIN.R30.EK1122_PortD_MissingLink
							OR (MAIN.R30.WS[1].ECatSlave_Cable_Breaks<>0) OR (MAIN.R30.WS[2].ECatSlave_Cable_Breaks<>0));
		Out_To_ICxx.System_Faults[900]:=Fault_Tmrs[900].Q;

	(*----- EOAT Cable(s) -------*)
	(*Fault901 - EOAT01 Cable(s) disconnected*)
		Fault_Tmrs[901].PT:=No_Timer;
		Fault_Tmrs[901]();
		Fault_Tmrs[901].IN:= (MAIN.R1.FB_In.Options.EOAT_Amount>=1) AND
							((EOAT01.ECatSlave_Cable_Breaks[0]<>0)
								OR (EOAT01.ECatSlave_Cable_Breaks[1]<>0));
		Out_To_ICxx.System_Faults[901]:=Fault_Tmrs[901].Q;
	(*Fault902 - EOAT02 Cable(s) disconnected*)
		Fault_Tmrs[902].PT:=No_Timer;
		Fault_Tmrs[902]();
		Fault_Tmrs[902].IN:= (MAIN.R2.FB_In.Options.EOAT_Amount>=2) AND
							((EOAT02.ECatSlave_Cable_Breaks[0]<>0)
								OR (EOAT02.ECatSlave_Cable_Breaks[1]<>0));
		Out_To_ICxx.System_Faults[902]:=Fault_Tmrs[902].Q;
	(*Fault903 - EOAT03 Cable(s) disconnected*)
		Fault_Tmrs[903].PT:=No_Timer;
		Fault_Tmrs[903]();
		Fault_Tmrs[903].IN:= (MAIN.R3.FB_In.Options.EOAT_Amount>=3) AND
							((EOAT04.ECatSlave_Cable_Breaks[0]<>0)
								OR (EOAT04.ECatSlave_Cable_Breaks[1]<>0));
		Out_To_ICxx.System_Faults[903]:=Fault_Tmrs[903].Q;
	(*Fault904 - EOAT04 Cable(s) disconnected*)
		Fault_Tmrs[904].PT:=No_Timer;
		Fault_Tmrs[904]();
		Fault_Tmrs[904].IN:= (MAIN.R4.FB_In.Options.EOAT_Amount>=4) AND
							((EOAT05.ECatSlave_Cable_Breaks[0]<>0)
								OR (EOAT05.ECatSlave_Cable_Breaks[1]<>0));
		Out_To_ICxx.System_Faults[904]:=Fault_Tmrs[904].Q;
	(*Fault905 - EOAT05 Cable(s) disconnected*)
		Fault_Tmrs[905].PT:=No_Timer;
		Fault_Tmrs[905]();
		Fault_Tmrs[905].IN:= (MAIN.R5.FB_In.Options.EOAT_Amount>=5) AND
							((EOAT05.ECatSlave_Cable_Breaks[0]<>0)
								OR (EOAT05.ECatSlave_Cable_Breaks[1]<>0));
		Out_To_ICxx.System_Faults[905]:=Fault_Tmrs[905].Q;
	(*Fault906 - EOAT06 Cable(s) disconnected*)
		Fault_Tmrs[906].PT:=No_Timer;
		Fault_Tmrs[906]();
		Fault_Tmrs[906].IN:= (MAIN.R6.FB_In.Options.EOAT_Amount>=6) AND
							((EOAT06.ECatSlave_Cable_Breaks[0]<>0)
								OR (EOAT06.ECatSlave_Cable_Breaks[1]<>0));
		Out_To_ICxx.System_Faults[906]:=Fault_Tmrs[906].Q;
	(*Fault907 - EOAT07 Cable(s) disconnected*)
		Fault_Tmrs[907].PT:=No_Timer;
		Fault_Tmrs[907]();
		Fault_Tmrs[907].IN:= (MAIN.R7.FB_In.Options.EOAT_Amount>=7) AND
							((EOAT07.ECatSlave_Cable_Breaks[0]<>0)
								OR (EOAT07.ECatSlave_Cable_Breaks[1]<>0));
		Out_To_ICxx.System_Faults[907]:=Fault_Tmrs[907].Q;
	(*Fault908 - EOAT08 Cable(s) disconnected*)
		Fault_Tmrs[908].PT:=No_Timer;
		Fault_Tmrs[908]();
		Fault_Tmrs[908].IN:= (MAIN.R8.FB_In.Options.EOAT_Amount>=8) AND
							((EOAT08.ECatSlave_Cable_Breaks[0]<>0)
								OR (EOAT08.ECatSlave_Cable_Breaks[1]<>0));
		Out_To_ICxx.System_Faults[908]:=Fault_Tmrs[908].Q;
	(*Fault909 - EOAT09 Cable(s) disconnected*)
		Fault_Tmrs[909].PT:=No_Timer;
		Fault_Tmrs[909]();
		Fault_Tmrs[909].IN:= (MAIN.R9.FB_In.Options.EOAT_Amount>=9) AND
							((EOAT09.ECatSlave_Cable_Breaks[0]<>0)
								OR (EOAT09.ECatSlave_Cable_Breaks[1]<>0));
		Out_To_ICxx.System_Faults[909]:=Fault_Tmrs[909].Q;
	(*Fault910 - EOAT10 Cable(s) disconnected*)
		Fault_Tmrs[820].PT:=No_Timer;
		Fault_Tmrs[820]();
		Fault_Tmrs[820].IN:=(MAIN.R10.FB_In.Options.EOAT_Amount>=10) AND
							((EOAT10.ECatSlave_Cable_Breaks[0]<>0)
								OR (EOAT10.ECatSlave_Cable_Breaks[1]<>0));
		Out_To_ICxx.System_Faults[820]:=Fault_Tmrs[820].Q; 
	(*Fault911 - EOAT11 Cable(s) disconnected*)
		Fault_Tmrs[911].PT:=No_Timer;
		Fault_Tmrs[911]();
		Fault_Tmrs[911].IN:= FALSE;
		Out_To_ICxx.System_Faults[911]:=Fault_Tmrs[911].Q;
	(*Fault912 - EOAT12 Cable(s) disconnected*)
		Fault_Tmrs[912].PT:=No_Timer;
		Fault_Tmrs[912]();
		Fault_Tmrs[912].IN:= FALSE;
		Out_To_ICxx.System_Faults[912]:=Fault_Tmrs[912].Q;
	(*Fault913 - EOAT13 Cable(s) disconnected*)
		Fault_Tmrs[913].PT:=No_Timer;
		Fault_Tmrs[913]();
		Fault_Tmrs[913].IN:= FALSE;
		Out_To_ICxx.System_Faults[913]:=Fault_Tmrs[913].Q;
	(*Fault914 - EOAT14 Cable(s) disconnected*)
		Fault_Tmrs[914].PT:=No_Timer;
		Fault_Tmrs[914]();
		Fault_Tmrs[914].IN:= FALSE;
		Out_To_ICxx.System_Faults[914]:=Fault_Tmrs[914].Q;
	(*Fault915 - EOAT15 Cable(s) disconnected*)
		Fault_Tmrs[915].PT:=No_Timer;
		Fault_Tmrs[915]();
		Fault_Tmrs[915].IN:= FALSE;
		Out_To_ICxx.System_Faults[915]:=Fault_Tmrs[915].Q;
	(*Fault916 - EOAT16 Cable(s) disconnected*)
		Fault_Tmrs[916].PT:=No_Timer;
		Fault_Tmrs[916]();
		Fault_Tmrs[916].IN:= FALSE;
		Out_To_ICxx.System_Faults[916]:=Fault_Tmrs[916].Q;
	(*Fault917 - EOAT17 Cable(s) disconnected*)
		Fault_Tmrs[917].PT:=No_Timer;
		Fault_Tmrs[917]();
		Fault_Tmrs[917].IN:= FALSE;
		Out_To_ICxx.System_Faults[917]:=Fault_Tmrs[917].Q;
	(*Fault918 - EOAT18 Cable(s) disconnected*)
		Fault_Tmrs[918].PT:=No_Timer;
		Fault_Tmrs[918]();
		Fault_Tmrs[918].IN:= FALSE;
		Out_To_ICxx.System_Faults[918]:=Fault_Tmrs[918].Q;
	(*Fault919 - EOAT19 Cable(s) disconnected*)
		Fault_Tmrs[919].PT:=No_Timer;
		Fault_Tmrs[919]();
		Fault_Tmrs[919].IN:= FALSE;
		Out_To_ICxx.System_Faults[919]:=Fault_Tmrs[919].Q;
	(*Fault920 - EOAT20 Cable(s) disconnected*)
		Fault_Tmrs[920].PT:=No_Timer;
		Fault_Tmrs[920]();
		Fault_Tmrs[920].IN:= FALSE;
		Out_To_ICxx.System_Faults[920]:=Fault_Tmrs[920].Q;
	(*Fault921 - EOAT21 Cable(s) disconnected*)
		Fault_Tmrs[921].PT:=No_Timer;
		Fault_Tmrs[921]();
		Fault_Tmrs[921].IN:= FALSE;
		Out_To_ICxx.System_Faults[921]:=Fault_Tmrs[921].Q;
	(*Fault922 - EOAT22 Cable(s) disconnected*)
		Fault_Tmrs[922].PT:=No_Timer;
		Fault_Tmrs[922]();
		Fault_Tmrs[922].IN:= FALSE;
		Out_To_ICxx.System_Faults[922]:=Fault_Tmrs[922].Q;
	(*Fault923 - EOAT23 Cable(s) disconnected*)
		Fault_Tmrs[923].PT:=No_Timer;
		Fault_Tmrs[923]();
		Fault_Tmrs[923].IN:= FALSE;
		Out_To_ICxx.System_Faults[923]:=Fault_Tmrs[923].Q;
	(*Fault924 - EOAT24 Cable(s) disconnected*)
		Fault_Tmrs[924].PT:=No_Timer;
		Fault_Tmrs[924]();
		Fault_Tmrs[924].IN:= FALSE;
		Out_To_ICxx.System_Faults[924]:=Fault_Tmrs[924].Q;
	(*Fault925 - EOAT25 Cable(s) disconnected*)
		Fault_Tmrs[925].PT:=No_Timer;
		Fault_Tmrs[925]();
		Fault_Tmrs[925].IN:= FALSE;
		Out_To_ICxx.System_Faults[925]:=Fault_Tmrs[925].Q;
	(*Fault926 - EOAT26 Cable(s) disconnected*)
		Fault_Tmrs[926].PT:=No_Timer;
		Fault_Tmrs[926]();
		Fault_Tmrs[926].IN:= FALSE;
		Out_To_ICxx.System_Faults[926]:=Fault_Tmrs[926].Q;
	(*Fault927 - EOAT27 Cable(s) disconnected*)
		Fault_Tmrs[927].PT:=No_Timer;
		Fault_Tmrs[927]();
		Fault_Tmrs[927].IN:= FALSE;
		Out_To_ICxx.System_Faults[927]:=Fault_Tmrs[927].Q;
	(*Fault928 - EOAT28 Cable(s) disconnected*)
		Fault_Tmrs[928].PT:=No_Timer;
		Fault_Tmrs[928]();
		Fault_Tmrs[928].IN:= FALSE;
		Out_To_ICxx.System_Faults[928]:=Fault_Tmrs[928].Q;
	(*Fault929 - EOAT29 Cable(s) disconnected*)
		Fault_Tmrs[929].PT:=No_Timer;
		Fault_Tmrs[929]();
		Fault_Tmrs[929].IN:= FALSE;
		Out_To_ICxx.System_Faults[929]:=Fault_Tmrs[929].Q;
	(*Fault930 - EOAT30 Cable(s) disconnected*)
		Fault_Tmrs[930].PT:=No_Timer;
		Fault_Tmrs[930]();
		Fault_Tmrs[930].IN:= FALSE;
		Out_To_ICxx.System_Faults[930]:=Fault_Tmrs[930].Q;


	(* --------------------------Services Stand Cable Faults----------------------------*)
	(*Fault931 - SS01 IN Cable Fault*)
		Fault_Tmrs[931].PT:=No_Timer;
		Fault_Tmrs[931]();
		Fault_Tmrs[931].IN:= GTAC_CONFIG.Option_Air1  AND
							MAIN.SS01.EP2028_NotPresent;
		Out_To_ICxx.System_Faults[931]:=Fault_Tmrs[931].Q;
	(*Fault932 - SS01 OUT Cable Fault*)
		Fault_Tmrs[932].PT:=No_Timer;
		Fault_Tmrs[932]();
		Fault_Tmrs[932].IN:= GTAC_CONFIG.Option_Air1  AND
							MAIN.SS01.EP1008_PortB_MissingLink;
		Out_To_ICxx.System_Faults[932]:=Fault_Tmrs[932].Q;
	(*Fault933 - SS02 IN Cable Fault*)
		Fault_Tmrs[933].PT:=No_Timer;
		Fault_Tmrs[933]();
		Fault_Tmrs[933].IN:= GTAC_CONFIG.Option_Air2  AND
							MAIN.SS02.EP2028_NotPresent;
		Out_To_ICxx.System_Faults[933]:=Fault_Tmrs[933].Q;
	(*Fault934 - SS02 OUT Cable Fault*)
		Fault_Tmrs[934].PT:=No_Timer;
		Fault_Tmrs[934]();
		Fault_Tmrs[934].IN:= GTAC_CONFIG.Option_Air2  AND
							MAIN.SS02.EP1008_PortB_MissingLink;
		Out_To_ICxx.System_Faults[934]:=Fault_Tmrs[934].Q;
(*
	(*Fault935 - SS03 IN Cable Fault*)
		Fault_Tmrs[935].PT:=No_Timer;
		Fault_Tmrs[935]();
		Fault_Tmrs[935].IN:= (GTAC_CONFIG.Option_Air1>=1)  AND
							MAIN.SS03.EP2028_NotPresent;
		Out_To_ICxx.System_Faults[935]:=Fault_Tmrs[935].Q;
	(*Fault936 - SS03 OUT Cable Fault*)
		Fault_Tmrs[936].PT:=No_Timer;
		Fault_Tmrs[936]();
		Fault_Tmrs[936].IN:= (GTAC_CONFIG.Option_Air1>=1)  AND
							MAIN.SS03.EP1008_PortB_MissingLink;
		Out_To_ICxx.System_Faults[936]:=Fault_Tmrs[546].Q;
*)
	(* --------------------------Enable Switch Plate Cable Faults----------------------------*)
	(*Fault937 - ESW01 IN Cable Fault*)
		Fault_Tmrs[937].PT:=No_Timer;
		Fault_Tmrs[937]();
		Fault_Tmrs[937].IN:= (GTAC_CONFIG.Option_ESW_Count>=1)  AND
							MAIN.ESW01.EP1908_NotPresent;
		Out_To_ICxx.System_Faults[937]:=Fault_Tmrs[937].Q;
	(*Fault938 - ESW01 OUT Cable Fault*)
		Fault_Tmrs[938].PT:=No_Timer;
		Fault_Tmrs[938]();
		Fault_Tmrs[938].IN:= (GTAC_CONFIG.Option_ESW_Count>=1)  AND
							MAIN.ESW01.EP1908_PortB_MissingLink;
		Out_To_ICxx.System_Faults[938]:=Fault_Tmrs[938].Q;
	(*Fault939 - ESW02 IN Cable Fault*)
		Fault_Tmrs[939].PT:=No_Timer;
		Fault_Tmrs[939]();
		Fault_Tmrs[939].IN:= (GTAC_CONFIG.Option_ESW_Count>=2)  AND
							MAIN.ESW02.EP1908_NotPresent;
		Out_To_ICxx.System_Faults[939]:=Fault_Tmrs[939].Q;
	(*Fault940 - ESW02 OUT Cable Fault*)
		Fault_Tmrs[940].PT:=No_Timer;
		Fault_Tmrs[940]();
		Fault_Tmrs[940].IN:= (GTAC_CONFIG.Option_ESW_Count>=2)  AND
							MAIN.ESW02.EP1908_PortB_MissingLink;
		Out_To_ICxx.System_Faults[940]:=Fault_Tmrs[940].Q;
	(*Fault941 - ESW03 IN Cable Fault*)
		Fault_Tmrs[941].PT:=No_Timer;
		Fault_Tmrs[941]();
		Fault_Tmrs[941].IN:= (GTAC_CONFIG.Option_ESW_Count>=3)  AND
							MAIN.ESW03.EP1908_NotPresent;
		Out_To_ICxx.System_Faults[941]:=Fault_Tmrs[941].Q;
	(*Fault942 - ESW03 OUT Cable Fault*)
		Fault_Tmrs[942].PT:=No_Timer;
		Fault_Tmrs[942]();
		Fault_Tmrs[942].IN:= (GTAC_CONFIG.Option_ESW_Count>=3)  AND
							MAIN.ESW03.EP1908_PortB_MissingLink;
		Out_To_ICxx.System_Faults[942]:=Fault_Tmrs[942].Q;
	(*Fault943 - ESW04 IN Cable Fault*)
		Fault_Tmrs[943].PT:=No_Timer;
		Fault_Tmrs[943]();
		Fault_Tmrs[943].IN:= (GTAC_CONFIG.Option_ESW_Count>=4)  AND
							MAIN.ESW04.EP1908_NotPresent;
		Out_To_ICxx.System_Faults[943]:=Fault_Tmrs[943].Q;
	(*Fault944 - ESW04 OUT Cable Fault*)
		Fault_Tmrs[944].PT:=No_Timer;
		Fault_Tmrs[944]();
		Fault_Tmrs[944].IN:= (GTAC_CONFIG.Option_ESW_Count>=4)  AND
							MAIN.ESW04.EP1908_PortB_MissingLink;
		Out_To_ICxx.System_Faults[944]:=Fault_Tmrs[944].Q;

(* -------------------------- IS Cable Faults----------------------------*)

	(*Fault751 - IS01 Cable break fault (any cable break)*)
		Fault_Tmrs[945].PT:= No_Timer;
		Fault_Tmrs[945]();
		Fault_Tmrs[945].IN:= (GTAC_CONFIG.Option_IS_Count >= 1) AND 
							(MAIN.IS01.ECatSlave_Cable_Breaks <> 0);
		Out_To_ICxx.System_Faults[945]:=Fault_Tmrs[945].Q;
	(*Fault752 - IS01 Profibus Network Fault*)
		Fault_Tmrs[946].PT:= No_Timer;
		Fault_Tmrs[946]();
		Fault_Tmrs[946].IN:= (GTAC_CONFIG.Option_IS_Count >= 1) AND 
							MAIN.IS01.FB_In.Option_Enable_Pbus AND
							NOT (MAIN.IS01.ProfiNode_OK);
		Out_To_ICxx.System_Faults[946]:=Fault_Tmrs[946].Q;

	(* -------------------------- Servo Drive Cable Faults----------------------------*)

